LIN {X 0,Y 249.09,Z 614.452,A -85,B 0,C 180,E1 -19011.52,E2 -19011.52} C_VEL
LIN {X 0,Y 249.134,Z 614.451,A -85,B 0,C 180,E1 -19015.483,E2 -19015.483} C_VEL
LIN {X 0,Y 249.086,Z 614.457,A -85,B 0,C 180,E1 -19018.994,E2 -19018.994} C_VEL
LIN {X 0,Y 249.034,Z 614.454,A -85,B 0,C 180,E1 -19022.427,E2 -19022.427} C_VEL
LIN {X 0,Y 249.033,Z 614.454,A -85,B 0,C 180,E1 -19026.347,E2 -19026.347} C_VEL
LIN {X 0,Y 249.01,Z 614.463,A -85,B 0,C 180,E1 -19030.479,E2 -19030.479} C_VEL
LIN {X 0,Y 249.012,Z 614.464,A -85,B 0,C 180,E1 -19034.879,E2 -19034.879} C_VEL
LIN {X 0,Y 249.023,Z 614.461,A -85,B 0,C 180,E1 -19037.364,E2 -19037.364} C_VEL
LIN {X 0,Y 249.048,Z 614.442,A -85,B 0,C 180,E1 -19042.201,E2 -19042.201} C_VEL
LIN {X 0,Y 249.062,Z 614.452,A -85,B 0,C 180,E1 -19045.642,E2 -19045.642} C_VEL
LIN {X 0,Y 249.058,Z 614.459,A -85,B 0,C 180,E1 -19049.474,E2 -19049.474} C_VEL
LIN {X 0,Y 249.076,Z 614.457,A -85,B 0,C 180,E1 -19053.163,E2 -19053.163} C_VEL
LIN {X 0,Y 249.067,Z 614.455,A -85,B 0,C 180,E1 -19056.732,E2 -19056.732} C_VEL
LIN {X 0,Y 249.114,Z 614.444,A -85,B 0,C 180,E1 -19060.212,E2 -19060.212} C_VEL
LIN {X 0,Y 249.229,Z 614.424,A -85,B 0,C 180,E1 -19063.621,E2 -19063.621} C_VEL
LIN {X 0,Y 249.251,Z 614.432,A -85,B 0,C 180,E1 -19068.617,E2 -19068.617} C_VEL
LIN {X 0,Y 249.461,Z 614.411,A -85,B 0,C 180,E1 -19071.902,E2 -19071.902} C_VEL
LIN {X 0,Y 249.302,Z 614.427,A -85,B 0,C 180,E1 -19075.149,E2 -19075.149} C_VEL
LIN {X 0,Y 249.682,Z 614.378,A -85,B 0,C 180,E1 -19078.387,E2 -19078.387} C_VEL
LIN {X 0,Y 249.682,Z 614.371,A -85,B 0,C 180,E1 -19081.613,E2 -19081.613} C_VEL
LIN {X 0,Y 249.46,Z 614.411,A -85,B 0,C 180,E1 -19086.471,E2 -19086.471} C_VEL
LIN {X 0,Y 249.35,Z 614.423,A -85,B 0,C 180,E1 -19089.736,E2 -19089.736} C_VEL
LIN {X 0,Y 249.208,Z 614.436,A -85,B 0,C 180,E1 -19093.176,E2 -19093.176} C_VEL
LIN {X 0,Y 248.455,Z 614.531,A -85,B 0,C 180,E1 -19094.523,E2 -19094.523} C_VEL
LIN {X 0,Y 245.512,Z 614.901,A -85,B 0,C 180,E1 -19096.719,E2 -19096.719} C_VEL
LIN {X 0,Y 243.082,Z 615.206,A -85,B 0,C 180,E1 -19098.507,E2 -19098.507} C_VEL
LIN {X 0,Y 242.083,Z 615.329,A -85,B 0,C 180,E1 -19099.896,E2 -19099.896} C_VEL
LIN {X 0,Y 242.022,Z 615.339,A -85,B 0,C 180,E1 -19100.366,E2 -19100.366} C_VEL
LIN {X 0,Y 242.047,Z 615.332,A -85,B 0,C 180,E1 -19103.985,E2 -19103.985} C_VEL
LIN {X 0,Y 242.014,Z 615.337,A -85,B 0,C 180,E1 -19107.687,E2 -19107.687} C_VEL
LIN {X 0,Y 241.981,Z 615.34,A -85,B 0,C 180,E1 -19111.52,E2 -19111.52} C_VEL
LIN {X 0,Y 242.012,Z 615.337,A -85,B 0,C 180,E1 -19115.596,E2 -19115.596} C_VEL
LIN {X 0,Y 241.962,Z 615.344,A -85,B 0,C 180,E1 -19119.718,E2 -19119.718} C_VEL
LIN {X 0,Y 241.94,Z 615.348,A -85,B 0,C 180,E1 -19124.2,E2 -19124.2} C_VEL
LIN {X 0,Y 241.945,Z 615.346,A -85,B 0,C 180,E1 -19128.077,E2 -19128.077} C_VEL
LIN {X 0,Y 242.052,Z 615.51,A -85,B 0,C 180,E1 -19132.427,E2 -19132.427} C_VEL
LIN {X 0,Y 244.646,Z 627.471,A -85,B 0,C 180,E1 -19136.918,E2 -19136.918} C_VEL
LIN {X 0,Y 246.406,Z 636.286,A -85,B 0,C 180,E1 -19140.064,E2 -19140.064} C_VEL
LIN {X 0,Y 249.038,Z 644.626,A -85,B 0,C 180,E1 -19140.629,E2 -19140.629} C_VEL
LIN {X 0,Y 254.197,Z 690.653,A -85,B 0,C 180,E1 -19142.772,E2 -19142.772} C_VEL
LIN {X 0,Y 251.927,Z 745.701,A -85,B 0,C 180,E1 -19144.655,E2 -19144.655} C_VEL
LIN {X 0,Y 250.918,Z 759.315,A -85,B 0,C 180,E1 -19145.431,E2 -19145.431} C_VEL
LIN {X 0,Y 249.494,Z 771.741,A -85,B 0,C 180,E1 -19146.442,E2 -19146.442} C_VEL
LIN {X 0,Y 247.996,Z 783.383,A -85,B 0,C 180,E1 -19147.724,E2 -19147.724} C_VEL
LIN {X 0,Y 246.379,Z 794.75,A -85,B 0,C 180,E1 -19149.327,E2 -19149.327} C_VEL
LIN {X 0,Y 244.853,Z 805.07,A -85,B 0,C 180,E1 -19151.159,E2 -19151.159} C_VEL
LIN {X 0,Y 243.381,Z 814.349,A -85,B 0,C 180,E1 -19153.214,E2 -19153.214} C_VEL
LIN {X 0,Y 242.001,Z 823.396,A -85,B 0,C 180,E1 -19155.707,E2 -19155.707} C_VEL
LIN {X 0,Y 240.951,Z 830.593,A -85,B 0,C 180,E1 -19158.217,E2 -19158.217} C_VEL
LIN {X 0,Y 240.406,Z 836.316,A -85,B 0,C 180,E1 -19160.746,E2 -19160.746} C_VEL
LIN {X 0,Y 240.177,Z 840.763,A -85,B 0,C 180,E1 -19163.277,E2 -19163.277} C_VEL
LIN {X 0,Y 240.138,Z 843.082,A -85,B 0,C 180,E1 -19164.961,E2 -19164.961} C_VEL
LIN {X 0,Y 240.121,Z 844.923,A -85,B 0,C 180,E1 -19166.642,E2 -19166.642} C_VEL
LIN {X 0,Y 240.106,Z 846.259,A -85,B 0,C 180,E1 -19168.321,E2 -19168.321} C_VEL
LIN {X 0,Y 240.181,Z 847.174,A -85,B 0,C 180,E1 -19169.998,E2 -19169.998} C_VEL
LIN {X 0,Y 240.065,Z 847.656,A -85,B 0,C 180,E1 -19171.676,E2 -19171.676} C_VEL
LIN {X 0,Y 240,Z 847.701,A -85,B 0,C 180,E1 -19173.356,E2 -19173.356} C_VEL
LIN {X 0,Y 239.982,Z 846.513,A -85,B 0,C 180,E1 -19176.725,E2 -19176.725} C_VEL
LIN {X 0,Y 240.174,Z 845.328,A -85,B 0,C 180,E1 -19178.411,E2 -19178.411} C_VEL
LIN {X 0,Y 240.765,Z 842.736,A -85,B 0,C 180,E1 -19180.936,E2 -19180.936} C_VEL
LIN {X 0,Y 241.698,Z 839.154,A -85,B 0,C 180,E1 -19183.449,E2 -19183.449} C_VEL
LIN {X 0,Y 243.307,Z 834.5,A -85,B 0,C 180,E1 -19185.925,E2 -19185.925} C_VEL
LIN {X 0,Y 245.188,Z 828.664,A -85,B 0,C 180,E1 -19188.377,E2 -19188.377} C_VEL
LIN {X 0,Y 247.548,Z 821.5,A -85,B 0,C 180,E1 -19190.784,E2 -19190.784} C_VEL
LIN {X 0,Y 250.481,Z 812.616,A -85,B 0,C 180,E1 -19193.128,E2 -19193.128} C_VEL
LIN {X 0,Y 253.214,Z 803.619,A -85,B 0,C 180,E1 -19195.039,E2 -19195.039} C_VEL
LIN {X 0,Y 256.378,Z 792.642,A -85,B 0,C 180,E1 -19196.89,E2 -19196.89} C_VEL
LIN {X 0,Y 259.194,Z 781.744,A -85,B 0,C 180,E1 -19198.325,E2 -19198.325} C_VEL
LIN {X 0,Y 261.882,Z 769.864,A -85,B 0,C 180,E1 -19199.544,E2 -19199.544} C_VEL
LIN {X 0,Y 264.132,Z 757.818,A -85,B 0,C 180,E1 -19200.476,E2 -19200.476} C_VEL
LIN {X 0,Y 265.875,Z 744.095,A -85,B 0,C 180,E1 -19201.247,E2 -19201.247} C_VEL
LIN {X 0,Y 267.554,Z 722.588,A -85,B 0,C 180,E1 -19202.004,E2 -19202.004} C_VEL
LIN {X 0,Y 269.546,Z 692.623,A -85,B 0,C 180,E1 -19203.018,E2 -19203.018} C_VEL
LIN {X 0,Y 268.044,Z 675.513,A -85,B 0,C 180,E1 -19204.173,E2 -19204.173} C_VEL
LIN {X 0,Y 266.933,Z 667.783,A -85,B 0,C 180,E1 -19204.815,E2 -19204.815} C_VEL
LIN {X 0,Y 261.946,Z 656.396,A -85,B 0,C 180,E1 -19206.616,E2 -19206.616} C_VEL
LIN {X 0,Y 256.701,Z 646.257,A -85,B 0,C 180,E1 -19208.625,E2 -19208.625} C_VEL
LIN {X 0,Y 253.564,Z 640.832,A -85,B 0,C 180,E1 -19209.927,E2 -19209.927} C_VEL
LIN {X 0,Y 250.312,Z 635.27,A -85,B 0,C 180,E1 -19211.38,E2 -19211.38} C_VEL
LIN {X 0,Y 246.826,Z 629.984,A -85,B 0,C 180,E1 -19213.06,E2 -19213.06} C_VEL
LIN {X 0,Y 246.403,Z 629.005,A -85,B 0,C 180,E1 -19213.361,E2 -19213.361} C_VEL
LIN {X 0,Y 244.701,Z 623.368,A -85,B 0,C 180,E1 -19217.551,E2 -19217.551} C_VEL
LIN {X 0,Y 243.332,Z 619.435,A -85,B 0,C 180,E1 -19221.241,E2 -19221.241} C_VEL
LIN {X 0,Y 243.018,Z 618.149,A -85,B 0,C 180,E1 -19222.604,E2 -19222.604} C_VEL
LIN {X 0,Y 241.985,Z 615.336,A -85,B 0,C 180,E1 -19226.508,E2 -19226.508} C_VEL
LIN {X 0,Y 242.007,Z 615.332,A -85,B 0,C 180,E1 -19230.596,E2 -19230.596} C_VEL
LIN {X 0,Y 242.061,Z 615.323,A -85,B 0,C 180,E1 -19234.182,E2 -19234.182} C_VEL
LIN {X 0,Y 242.047,Z 615.336,A -85,B 0,C 180,E1 -19238.296,E2 -19238.296} C_VEL
LIN {X 0,Y 242.156,Z 615.318,A -85,B 0,C 180,E1 -19243.277,E2 -19243.277} C_VEL
LIN {X 0,Y 242.191,Z 615.438,A -85,B 0,C 180,E1 -19247.216,E2 -19247.216} C_VEL
LIN {X 0,Y 243.204,Z 617.796,A -85,B 0,C 180,E1 -19250.433,E2 -19250.433} C_VEL
LIN {X 0,Y 246.677,Z 622.197,A -85,B 0,C 180,E1 -19252.324,E2 -19252.324} C_VEL
LIN {X 0,Y 248.068,Z 623.799,A -85,B 0,C 180,E1 -19253.001,E2 -19253.001} C_VEL
LIN {X 0,Y 250.491,Z 627.155,A -85,B 0,C 180,E1 -19254.162,E2 -19254.162} C_VEL
LIN {X 0,Y 255.517,Z 633.633,A -85,B 0,C 180,E1 -19256.267,E2 -19256.267} C_VEL
LIN {X 0,Y 258.653,Z 638.212,A -85,B 0,C 180,E1 -19257.49,E2 -19257.49} C_VEL
LIN {X 0,Y 262.624,Z 644.888,A -85,B 0,C 180,E1 -19258.956,E2 -19258.956} C_VEL
LIN {X 0,Y 268.996,Z 656.761,A -85,B 0,C 180,E1 -19261.126,E2 -19261.126} C_VEL
LIN {X 0,Y 271.338,Z 662.521,A -85,B 0,C 180,E1 -19261.936,E2 -19261.936} C_VEL
LIN {X 0,Y 267.251,Z 720.175,A -85,B 0,C 180,E1 -19263.904,E2 -19263.904} C_VEL
LIN {X 0,Y 265.754,Z 733.662,A -85,B 0,C 180,E1 -19264.645,E2 -19264.645} C_VEL
LIN {X 0,Y 263.976,Z 746.003,A -85,B 0,C 180,E1 -19265.634,E2 -19265.634} C_VEL
LIN {X 0,Y 261.538,Z 758.402,A -85,B 0,C 180,E1 -19266.954,E2 -19266.954} C_VEL
LIN {X 0,Y 258.731,Z 770.225,A -85,B 0,C 180,E1 -19268.592,E2 -19268.592} C_VEL
LIN {X 0,Y 256.044,Z 780.215,A -85,B 0,C 180,E1 -19270.375,E2 -19270.375} C_VEL
LIN {X 0,Y 253.014,Z 789.597,A -85,B 0,C 180,E1 -19272.431,E2 -19272.431} C_VEL
LIN {X 0,Y 250.307,Z 797.53,A -85,B 0,C 180,E1 -19274.637,E2 -19274.637} C_VEL
LIN {X 0,Y 247.9,Z 803.973,A -85,B 0,C 180,E1 -19276.893,E2 -19276.893} C_VEL
LIN {X 0,Y 245.756,Z 809.422,A -85,B 0,C 180,E1 -19279.321,E2 -19279.321} C_VEL
LIN {X 0,Y 243.88,Z 814.004,A -85,B 0,C 180,E1 -19282.001,E2 -19282.001} C_VEL
LIN {X 0,Y 242.823,Z 816.492,A -85,B 0,C 180,E1 -19283.904,E2 -19283.904} C_VEL
LIN {X 0,Y 241.896,Z 818.362,A -85,B 0,C 180,E1 -19285.836,E2 -19285.836} C_VEL
LIN {X 0,Y 240.806,Z 820.184,A -85,B 0,C 180,E1 -19288.893,E2 -19288.893} C_VEL
LIN {X 0,Y 240.157,Z 820.642,A -85,B 0,C 180,E1 -19291.938,E2 -19291.938} C_VEL
LIN {X 0,Y 239.883,Z 819.775,A -85,B 0,C 180,E1 -19294.886,E2 -19294.886} C_VEL
LIN {X 0,Y 239.936,Z 817.519,A -85,B 0,C 180,E1 -19297.96,E2 -19297.96} C_VEL
LIN {X 0,Y 240.273,Z 814.563,A -85,B 0,C 180,E1 -19300.495,E2 -19300.495} C_VEL
LIN {X 0,Y 240.812,Z 810.309,A -85,B 0,C 180,E1 -19303.149,E2 -19303.149} C_VEL
LIN {X 0,Y 241.706,Z 804.016,A -85,B 0,C 180,E1 -19306.093,E2 -19306.093} C_VEL
LIN {X 0,Y 242.861,Z 796.483,A -85,B 0,C 180,E1 -19308.798,E2 -19308.798} C_VEL
LIN {X 0,Y 244.104,Z 788.762,A -85,B 0,C 180,E1 -19311.019,E2 -19311.019} C_VEL
LIN {X 0,Y 245.628,Z 779.186,A -85,B 0,C 180,E1 -19313.239,E2 -19313.239} C_VEL
LIN {X 0,Y 247.171,Z 769.108,A -85,B 0,C 180,E1 -19315.118,E2 -19315.118} C_VEL
LIN {X 0,Y 248.769,Z 757.73,A -85,B 0,C 180,E1 -19316.819,E2 -19316.819} C_VEL
LIN {X 0,Y 250.155,Z 745.895,A -85,B 0,C 180,E1 -19318.196,E2 -19318.196} C_VEL
LIN {X 0,Y 251.352,Z 732.633,A -85,B 0,C 180,E1 -19319.37,E2 -19319.37} C_VEL
LIN {X 0,Y 252.214,Z 719.571,A -85,B 0,C 180,E1 -19320.175,E2 -19320.175} C_VEL
LIN {X 0,Y 253.12,Z 698.707,A -85,B 0,C 180,E1 -19320.949,E2 -19320.949} C_VEL
LIN {X 0,Y 255.107,Z 648.228,A -85,B 0,C 180,E1 -19322.633,E2 -19322.633} C_VEL
LIN {X 0,Y 249.56,Z 633.732,A -85,B 0,C 180,E1 -19323.648,E2 -19323.648} C_VEL
LIN {X 0,Y 242.276,Z 616.171,A -85,B 0,C 180,E1 -19325.014,E2 -19325.014} C_VEL
LIN {X 0,Y 242.084,Z 615.328,A -85,B 0,C 180,E1 -19325.107,E2 -19325.107} C_VEL
LIN {X 0,Y 242.059,Z 615.334,A -85,B 0,C 180,E1 -19329.612,E2 -19329.612} C_VEL
LIN {X 0,Y 242.161,Z 615.318,A -85,B 0,C 180,E1 -19333.28,E2 -19333.28} C_VEL
LIN {X 0,Y 242.187,Z 615.319,A -85,B 0,C 180,E1 -19338.282,E2 -19338.282} C_VEL
LIN {X 0,Y 242.435,Z 615.285,A -85,B 0,C 180,E1 -19341.668,E2 -19341.668} C_VEL
LIN {X 0,Y 242.262,Z 615.307,A -85,B 0,C 180,E1 -19345.009,E2 -19345.009} C_VEL
LIN {X 0,Y 242.638,Z 615.263,A -85,B 0,C 180,E1 -19348.342,E2 -19348.342} C_VEL
LIN {X 0,Y 242.641,Z 615.259,A -85,B 0,C 180,E1 -19351.662,E2 -19351.662} C_VEL
LIN {X 0,Y 242.436,Z 615.287,A -85,B 0,C 180,E1 -19356.661,E2 -19356.661} C_VEL
LIN {X 0,Y 242.348,Z 615.295,A -85,B 0,C 180,E1 -19360.022,E2 -19360.022} C_VEL
LIN {X 0,Y 242.17,Z 615.318,A -85,B 0,C 180,E1 -19365.142,E2 -19365.142} C_VEL
LIN {X 0,Y 242.076,Z 615.327,A -85,B 0,C 180,E1 -19368.626,E2 -19368.626} C_VEL
LIN {X 0,Y 242.016,Z 615.333,A -85,B 0,C 180,E1 -19372.181,E2 -19372.181} C_VEL
LIN {X 0,Y 242.07,Z 615.329,A -85,B 0,C 180,E1 -19375.84,E2 -19375.84} C_VEL
LIN {X 0,Y 242.034,Z 615.331,A -85,B 0,C 180,E1 -19379.582,E2 -19379.582} C_VEL
LIN {X 0,Y 241.984,Z 615.327,A -85,B 0,C 180,E1 -19383.494,E2 -19383.494} C_VEL
LIN {X 0,Y 241.99,Z 615.337,A -85,B 0,C 180,E1 -19387.584,E2 -19387.584} C_VEL
LIN {X 0,Y 241.943,Z 615.345,A -85,B 0,C 180,E1 -19391.923,E2 -19391.923} C_VEL
LIN {X 0,Y 241.942,Z 615.341,A -85,B 0,C 180,E1 -19396.572,E2 -19396.572} C_VEL
LIN {X 0,Y 241.961,Z 615.33,A -85,B 0,C 180,E1 -19400.282,E2 -19400.282} C_VEL
LIN {X 0,Y 242.01,Z 615.324,A -85,B 0,C 180,E1 -19404.493,E2 -19404.493} C_VEL
LIN {X 0,Y 241.981,Z 615.337,A -85,B 0,C 180,E1 -19408.481,E2 -19408.481} C_VEL
LIN {X 0,Y 242.013,Z 615.337,A -85,B 0,C 180,E1 -19412.314,E2 -19412.314} C_VEL
LIN {X 0,Y 242.047,Z 615.332,A -85,B 0,C 180,E1 -19416.015,E2 -19416.015} C_VEL
LIN {X 0,Y 242.041,Z 615.329,A -85,B 0,C 180,E1 -19419.608,E2 -19419.608} C_VEL
LIN {X 0,Y 242.17,Z 615.301,A -85,B 0,C 180,E1 -19423.279,E2 -19423.279} C_VEL
LIN {X 0,Y 242.187,Z 615.313,A -85,B 0,C 180,E1 -19428.28,E2 -19428.28} C_VEL
LIN {X 0,Y 242.407,Z 615.288,A -85,B 0,C 180,E1 -19431.665,E2 -19431.665} C_VEL
LIN {X 0,Y 242.262,Z 615.304,A -85,B 0,C 180,E1 -19435.007,E2 -19435.007} C_VEL
LIN {X 0,Y 242.642,Z 615.254,A -85,B 0,C 180,E1 -19438.34,E2 -19438.34} C_VEL
LIN {X 0,Y 242.642,Z 615.247,A -85,B 0,C 180,E1 -19441.66,E2 -19441.66} C_VEL
LIN {X 0,Y 242.431,Z 615.285,A -85,B 0,C 180,E1 -19446.659,E2 -19446.659} C_VEL
LIN {X 0,Y 242.274,Z 615.306,A -85,B 0,C 180,E1 -19450.024,E2 -19450.024} C_VEL
LIN {X 0,Y 242.134,Z 615.315,A -85,B 0,C 180,E1 -19455.143,E2 -19455.143} C_VEL
LIN {X 0,Y 242.049,Z 615.336,A -85,B 0,C 180,E1 -19458.626,E2 -19458.626} C_VEL
LIN {X 0,Y 242.022,Z 615.339,A -85,B 0,C 180,E1 -19460.366,E2 -19460.366} C_VEL
LIN {X 0,Y 241.4,Z 615.424,A -85,B 0,C 180,E1 -19461.756,E2 -19461.756} C_VEL
LIN {X 0,Y 238.534,Z 615.777,A -85,B 0,C 180,E1 -19464.02,E2 -19464.02} C_VEL
LIN {X 0,Y 236.07,Z 616.077,A -85,B 0,C 180,E1 -19465.866,E2 -19465.866} C_VEL
LIN {X 0,Y 235.015,Z 616.21,A -85,B 0,C 180,E1 -19467.3,E2 -19467.3} C_VEL
LIN {X 0,Y 234.933,Z 616.217,A -85,B 0,C 180,E1 -19467.786,E2 -19467.786} C_VEL
LIN {X 0,Y 234.938,Z 616.223,A -85,B 0,C 180,E1 -19470.567,E2 -19470.567} C_VEL
LIN {X 0,Y 234.936,Z 616.22,A -85,B 0,C 180,E1 -19474.637,E2 -19474.637} C_VEL
LIN {X 0,Y 234.948,Z 616.221,A -85,B 0,C 180,E1 -19478.944,E2 -19478.944} C_VEL
LIN {X 0,Y 234.896,Z 616.226,A -85,B 0,C 180,E1 -19483.484,E2 -19483.484} C_VEL
LIN {X 0,Y 234.896,Z 616.226,A -85,B 0,C 180,E1 -19486.514,E2 -19486.514} C_VEL
LIN {X 0,Y 234.958,Z 616.218,A -85,B 0,C 180,E1 -19491.633,E2 -19491.633} C_VEL
LIN {X 0,Y 234.992,Z 616.275,A -85,B 0,C 180,E1 -19491.912,E2 -19491.912} C_VEL
LIN {X 0,Y 237.244,Z 626.919,A -85,B 0,C 180,E1 -19496.044,E2 -19496.044} C_VEL
LIN {X 0,Y 239.128,Z 636.083,A -85,B 0,C 180,E1 -19499.38,E2 -19499.38} C_VEL
LIN {X 0,Y 242.507,Z 646.258,A -85,B 0,C 180,E1 -19500.104,E2 -19500.104} C_VEL
LIN {X 0,Y 247.472,Z 690.694,A -85,B 0,C 180,E1 -19502.25,E2 -19502.25} C_VEL
LIN {X 0,Y 245.129,Z 745.513,A -85,B 0,C 180,E1 -19504.185,E2 -19504.185} C_VEL
LIN {X 0,Y 244.097,Z 759.046,A -85,B 0,C 180,E1 -19504.982,E2 -19504.982} C_VEL
LIN {X 0,Y 242.579,Z 771.91,A -85,B 0,C 180,E1 -19506.069,E2 -19506.069} C_VEL
LIN {X 0,Y 240.9,Z 784.211,A -85,B 0,C 180,E1 -19507.484,E2 -19507.484} C_VEL
LIN {X 0,Y 239.249,Z 795.356,A -85,B 0,C 180,E1 -19509.133,E2 -19509.133} C_VEL
LIN {X 0,Y 237.565,Z 806.32,A -85,B 0,C 180,E1 -19511.205,E2 -19511.205} C_VEL
LIN {X 0,Y 235.958,Z 816.257,A -85,B 0,C 180,E1 -19513.561,E2 -19513.561} C_VEL
LIN {X 0,Y 234.646,Z 824.795,A -85,B 0,C 180,E1 -19516.135,E2 -19516.135} C_VEL
LIN {X 0,Y 233.751,Z 831.643,A -85,B 0,C 180,E1 -19518.728,E2 -19518.728} C_VEL
LIN {X 0,Y 233.253,Z 837.07,A -85,B 0,C 180,E1 -19521.333,E2 -19521.333} C_VEL
LIN {X 0,Y 233.101,Z 841.65,A -85,B 0,C 180,E1 -19524.244,E2 -19524.244} C_VEL
LIN {X 0,Y 233.058,Z 844.256,A -85,B 0,C 180,E1 -19526.54,E2 -19526.54} C_VEL
LIN {X 0,Y 233.033,Z 845.674,A -85,B 0,C 180,E1 -19528.27,E2 -19528.27} C_VEL
LIN {X 0,Y 233.101,Z 846.634,A -85,B 0,C 180,E1 -19529.998,E2 -19529.998} C_VEL
LIN {X 0,Y 232.99,Z 847.159,A -85,B 0,C 180,E1 -19531.727,E2 -19531.727} C_VEL
LIN {X 0,Y 232.911,Z 847.276,A -85,B 0,C 180,E1 -19533.458,E2 -19533.458} C_VEL
LIN {X 0,Y 232.841,Z 846.949,A -85,B 0,C 180,E1 -19535.193,E2 -19535.193} C_VEL
LIN {X 0,Y 233.115,Z 845.072,A -85,B 0,C 180,E1 -19538.668,E2 -19538.668} C_VEL
LIN {X 0,Y 233.497,Z 843.536,A -85,B 0,C 180,E1 -19540.402,E2 -19540.402} C_VEL
LIN {X 0,Y 234.375,Z 840.387,A -85,B 0,C 180,E1 -19542.995,E2 -19542.995} C_VEL
LIN {X 0,Y 235.862,Z 836.23,A -85,B 0,C 180,E1 -19545.554,E2 -19545.554} C_VEL
LIN {X 0,Y 238.069,Z 829.963,A -85,B 0,C 180,E1 -19548.501,E2 -19548.501} C_VEL
LIN {X 0,Y 240.479,Z 823.171,A -85,B 0,C 180,E1 -19550.976,E2 -19550.976} C_VEL
LIN {X 0,Y 243.4,Z 814.814,A -85,B 0,C 180,E1 -19553.39,E2 -19553.39} C_VEL
LIN {X 0,Y 246.324,Z 806.382,A -85,B 0,C 180,E1 -19555.337,E2 -19555.337} C_VEL
LIN {X 0,Y 249.175,Z 797.33,A -85,B 0,C 180,E1 -19557.05,E2 -19557.05} C_VEL
LIN {X 0,Y 252.318,Z 786.286,A -85,B 0,C 180,E1 -19558.714,E2 -19558.714} C_VEL
LIN {X 0,Y 255.444,Z 773.963,A -85,B 0,C 180,E1 -19560.137,E2 -19560.137} C_VEL
LIN {X 0,Y 257.869,Z 762.16,A -85,B 0,C 180,E1 -19561.184,E2 -19561.184} C_VEL
LIN {X 0,Y 260.109,Z 747.995,A -85,B 0,C 180,E1 -19562.078,E2 -19562.078} C_VEL
LIN {X 0,Y 261.579,Z 733.711,A -85,B 0,C 180,E1 -19562.668,E2 -19562.668} C_VEL
LIN {X 0,Y 264.451,Z 693.887,A -85,B 0,C 180,E1 -19564.042,E2 -19564.042} C_VEL
LIN {X 0,Y 263.15,Z 677.789,A -85,B 0,C 180,E1 -19565.166,E2 -19565.166} C_VEL
LIN {X 0,Y 262.152,Z 670.998,A -85,B 0,C 180,E1 -19565.763,E2 -19565.763} C_VEL
LIN {X 0,Y 257.876,Z 660.878,A -85,B 0,C 180,E1 -19567.44,E2 -19567.44} C_VEL
LIN {X 0,Y 253.124,Z 651.404,A -85,B 0,C 180,E1 -19569.386,E2 -19569.386} C_VEL
LIN {X 0,Y 250.3,Z 646.33,A -85,B 0,C 180,E1 -19570.626,E2 -19570.626} C_VEL
LIN {X 0,Y 247.149,Z 640.848,A -85,B 0,C 180,E1 -19572.12,E2 -19572.12} C_VEL
LIN {X 0,Y 243.758,Z 635.331,A -85,B 0,C 180,E1 -19573.879,E2 -19573.879} C_VEL
LIN {X 0,Y 239.537,Z 629.3,A -85,B 0,C 180,E1 -19576.337,E2 -19576.337} C_VEL
LIN {X 0,Y 238.846,Z 627.89,A -85,B 0,C 180,E1 -19576.833,E2 -19576.833} C_VEL
LIN {X 0,Y 237.669,Z 624.13,A -85,B 0,C 180,E1 -19580.246,E2 -19580.246} C_VEL
LIN {X 0,Y 236.654,Z 621.209,A -85,B 0,C 180,E1 -19583.562,E2 -19583.562} C_VEL
LIN {X 0,Y 236.001,Z 619.137,A -85,B 0,C 180,E1 -19586.49,E2 -19586.49} C_VEL
LIN {X 0,Y 235.092,Z 616.975,A -85,B 0,C 180,E1 -19591.424,E2 -19591.424} C_VEL
LIN {X 0,Y 235.008,Z 616.205,A -85,B 0,C 180,E1 -19594.882,E2 -19594.882} C_VEL
LIN {X 0,Y 235.005,Z 616.222,A -85,B 0,C 180,E1 -19598.969,E2 -19598.969} C_VEL
LIN {X 0,Y 235.286,Z 617.222,A -85,B 0,C 180,E1 -19602.902,E2 -19602.902} C_VEL
LIN {X 0,Y 236.092,Z 618.98,A -85,B 0,C 180,E1 -19606.716,E2 -19606.716} C_VEL
LIN {X 0,Y 238.744,Z 622.515,A -85,B 0,C 180,E1 -19608.646,E2 -19608.646} C_VEL
LIN {X 0,Y 241.151,Z 624.593,A -85,B 0,C 180,E1 -19610.07,E2 -19610.07} C_VEL
LIN {X 0,Y 244.476,Z 628.746,A -85,B 0,C 180,E1 -19611.944,E2 -19611.944} C_VEL
LIN {X 0,Y 246.301,Z 631.399,A -85,B 0,C 180,E1 -19612.89,E2 -19612.89} C_VEL
LIN {X 0,Y 249.219,Z 635.19,A -85,B 0,C 180,E1 -19614.278,E2 -19614.278} C_VEL
LIN {X 0,Y 252.66,Z 639.789,A -85,B 0,C 180,E1 -19615.755,E2 -19615.755} C_VEL
LIN {X 0,Y 256.339,Z 645.372,A -85,B 0,C 180,E1 -19617.262,E2 -19617.262} C_VEL
LIN {X 0,Y 263.166,Z 658.178,A -85,B 0,C 180,E1 -19619.842,E2 -19619.842} C_VEL
LIN {X 0,Y 266.218,Z 664.61,A -85,B 0,C 180,E1 -19620.898,E2 -19620.898} C_VEL
LIN {X 0,Y 261.994,Z 721.142,A -85,B 0,C 180,E1 -19622.892,E2 -19622.892} C_VEL
LIN {X 0,Y 260.338,Z 734.926,A -85,B 0,C 180,E1 -19623.678,E2 -19623.678} C_VEL
LIN {X 0,Y 258.256,Z 748.052,A -85,B 0,C 180,E1 -19624.78,E2 -19624.78} C_VEL
LIN {X 0,Y 255.739,Z 760.064,A -85,B 0,C 180,E1 -19626.113,E2 -19626.113} C_VEL
LIN {X 0,Y 253.124,Z 770.531,A -85,B 0,C 180,E1 -19627.601,E2 -19627.601} C_VEL
LIN {X 0,Y 250.474,Z 779.913,A -85,B 0,C 180,E1 -19629.284,E2 -19629.284} C_VEL
LIN {X 0,Y 247.79,Z 787.852,A -85,B 0,C 180,E1 -19630.996,E2 -19630.996} C_VEL
LIN {X 0,Y 244.723,Z 796.298,A -85,B 0,C 180,E1 -19633.282,E2 -19633.282} C_VEL
LIN {X 0,Y 242.025,Z 803.245,A -85,B 0,C 180,E1 -19635.642,E2 -19635.642} C_VEL
LIN {X 0,Y 239.771,Z 808.574,A -85,B 0,C 180,E1 -19637.925,E2 -19637.925} C_VEL
LIN {X 0,Y 237.577,Z 813.692,A -85,B 0,C 180,E1 -19640.792,E2 -19640.792} C_VEL
LIN {X 0,Y 235.837,Z 817.379,A -85,B 0,C 180,E1 -19643.721,E2 -19643.721} C_VEL
LIN {X 0,Y 234.434,Z 819.811,A -85,B 0,C 180,E1 -19646.723,E2 -19646.723} C_VEL
LIN {X 0,Y 233.621,Z 820.875,A -85,B 0,C 180,E1 -19649.265,E2 -19649.265} C_VEL
LIN {X 0,Y 233.004,Z 820.961,A -85,B 0,C 180,E1 -19652.38,E2 -19652.38} C_VEL
LIN {X 0,Y 232.763,Z 819.795,A -85,B 0,C 180,E1 -19655.393,E2 -19655.393} C_VEL
LIN {X 0,Y 232.882,Z 817.459,A -85,B 0,C 180,E1 -19658.316,E2 -19658.316} C_VEL
LIN {X 0,Y 233.364,Z 813.444,A -85,B 0,C 180,E1 -19661.495,E2 -19661.495} C_VEL
LIN {X 0,Y 233.925,Z 809.401,A -85,B 0,C 180,E1 -19663.862,E2 -19663.862} C_VEL
LIN {X 0,Y 234.848,Z 802.822,A -85,B 0,C 180,E1 -19666.837,E2 -19666.837} C_VEL
LIN {X 0,Y 235.979,Z 795.789,A -85,B 0,C 180,E1 -19669.331,E2 -19669.331} C_VEL
LIN {X 0,Y 237.396,Z 787.283,A -85,B 0,C 180,E1 -19671.737,E2 -19671.737} C_VEL
LIN {X 0,Y 239.019,Z 777.426,A -85,B 0,C 180,E1 -19673.982,E2 -19673.982} C_VEL
LIN {X 0,Y 240.657,Z 766.648,A -85,B 0,C 180,E1 -19675.943,E2 -19675.943} C_VEL
LIN {X 0,Y 242.216,Z 755.048,A -85,B 0,C 180,E1 -19677.611,E2 -19677.611} C_VEL
LIN {X 0,Y 243.677,Z 743.022,A -85,B 0,C 180,E1 -19678.958,E2 -19678.958} C_VEL
LIN {X 0,Y 244.871,Z 729.452,A -85,B 0,C 180,E1 -19680.079,E2 -19680.079} C_VEL
LIN {X 0,Y 245.655,Z 716,A -85,B 0,C 180,E1 -19680.846,E2 -19680.846} C_VEL
LIN {X 0,Y 248.481,Z 649.907,A -85,B 0,C 180,E1 -19683.13,E2 -19683.13} C_VEL
LIN {X 0,Y 242.604,Z 634.793,A -85,B 0,C 180,E1 -19684.246,E2 -19684.246} C_VEL
LIN {X 0,Y 235.172,Z 617.035,A -85,B 0,C 180,E1 -19685.681,E2 -19685.681} C_VEL
LIN {X 0,Y 235.026,Z 616.209,A -85,B 0,C 180,E1 -19685.783,E2 -19685.783} C_VEL
LIN {X 0,Y 235.026,Z 616.209,A -85,B 0,C 180,E1 -19688.973,E2 -19688.973} C_VEL
LIN {X 0,Y 235.095,Z 616.198,A -85,B 0,C 180,E1 -19693.061,E2 -19693.061} C_VEL
LIN {X 0,Y 235.147,Z 616.194,A -85,B 0,C 180,E1 -19697.926,E2 -19697.926} C_VEL
LIN {X 0,Y 235.39,Z 616.163,A -85,B 0,C 180,E1 -19701.416,E2 -19701.416} C_VEL
LIN {X 0,Y 235.406,Z 616.161,A -85,B 0,C 180,E1 -19703.143,E2 -19703.143} C_VEL
LIN {X 0,Y 235.597,Z 616.14,A -85,B 0,C 180,E1 -19708.292,E2 -19708.292} C_VEL
LIN {X 0,Y 235.6,Z 616.136,A -85,B 0,C 180,E1 -19711.711,E2 -19711.711} C_VEL
LIN {X 0,Y 235.408,Z 616.162,A -85,B 0,C 180,E1 -19716.86,E2 -19716.86} C_VEL
LIN {X 0,Y 235.256,Z 616.18,A -85,B 0,C 180,E1 -19720.328,E2 -19720.328} C_VEL
LIN {X 0,Y 235.117,Z 616.195,A -85,B 0,C 180,E1 -19725.608,E2 -19725.608} C_VEL
LIN {X 0,Y 235.012,Z 616.201,A -85,B 0,C 180,E1 -19729.207,E2 -19729.207} C_VEL
LIN {X 0,Y 234.964,Z 616.214,A -85,B 0,C 180,E1 -19732.884,E2 -19732.884} C_VEL
LIN {X 0,Y 234.973,Z 616.215,A -85,B 0,C 180,E1 -19736.659,E2 -19736.659} C_VEL
LIN {X 0,Y 234.935,Z 616.215,A -85,B 0,C 180,E1 -19740.569,E2 -19740.569} C_VEL
LIN {X 0,Y 234.931,Z 616.203,A -85,B 0,C 180,E1 -19744.64,E2 -19744.64} C_VEL
LIN {X 0,Y 234.946,Z 616.214,A -85,B 0,C 180,E1 -19748.946,E2 -19748.946} C_VEL
LIN {X 0,Y 234.894,Z 616.225,A -85,B 0,C 180,E1 -19753.487,E2 -19753.487} C_VEL
LIN {X 0,Y 234.895,Z 616.219,A -85,B 0,C 180,E1 -19756.516,E2 -19756.516} C_VEL
LIN {X 0,Y 234.923,Z 616.207,A -85,B 0,C 180,E1 -19761.08,E2 -19761.08} C_VEL
LIN {X 0,Y 234.947,Z 616.205,A -85,B 0,C 180,E1 -19765.365,E2 -19765.365} C_VEL
LIN {X 0,Y 234.938,Z 616.217,A -85,B 0,C 180,E1 -19769.433,E2 -19769.433} C_VEL
LIN {X 0,Y 235,Z 616.213,A -85,B 0,C 180,E1 -19773.795,E2 -19773.795} C_VEL
LIN {X 0,Y 235.004,Z 616.203,A -85,B 0,C 180,E1 -19778.969,E2 -19778.969} C_VEL
LIN {X 0,Y 235.102,Z 616.179,A -85,B 0,C 180,E1 -19783.061,E2 -19783.061} C_VEL
LIN {X 0,Y 235.12,Z 616.19,A -85,B 0,C 180,E1 -19787.923,E2 -19787.923} C_VEL
LIN {X 0,Y 235.338,Z 616.167,A -85,B 0,C 180,E1 -19791.413,E2 -19791.413} C_VEL
LIN {X 0,Y 235.38,Z 616.162,A -85,B 0,C 180,E1 -19793.141,E2 -19793.141} C_VEL
LIN {X 0,Y 235.602,Z 616.131,A -85,B 0,C 180,E1 -19798.291,E2 -19798.291} C_VEL
LIN {X 0,Y 235.602,Z 616.123,A -85,B 0,C 180,E1 -19801.71,E2 -19801.71} C_VEL
LIN {X 0,Y 235.381,Z 616.163,A -85,B 0,C 180,E1 -19806.86,E2 -19806.86} C_VEL
LIN {X 0,Y 235.221,Z 616.187,A -85,B 0,C 180,E1 -19810.327,E2 -19810.327} C_VEL
LIN {X 0,Y 235.081,Z 616.193,A -85,B 0,C 180,E1 -19815.609,E2 -19815.609} C_VEL
LIN {X 0,Y 234.966,Z 616.213,A -85,B 0,C 180,E1 -19820.375,E2 -19820.375} C_VEL
LIN {X 0,Y 234.985,Z 616.211,A -85,B 0,C 180,E1 -19824.754,E2 -19824.754} C_VEL
LIN {X 0,Y 234.933,Z 616.217,A -85,B 0,C 180,E1 -19827.786,E2 -19827.786} C_VEL
LIN {X 0,Y 234.261,Z 616.306,A -85,B 0,C 180,E1 -19829.216,E2 -19829.216} C_VEL
LIN {X 0,Y 231.367,Z 616.662,A -85,B 0,C 180,E1 -19831.547,E2 -19831.547} C_VEL
LIN {X 0,Y 228.93,Z 616.966,A -85,B 0,C 180,E1 -19833.448,E2 -19833.448} C_VEL
LIN {X 0,Y 227.922,Z 617.096,A -85,B 0,C 180,E1 -19834.925,E2 -19834.925} C_VEL
LIN {X 0,Y 227.86,Z 617.096,A -85,B 0,C 180,E1 -19835.426,E2 -19835.426} C_VEL
LIN {X 0,Y 227.859,Z 617.102,A -85,B 0,C 180,E1 -19839.545,E2 -19839.545} C_VEL
LIN {X 0,Y 227.819,Z 617.11,A -85,B 0,C 180,E1 -19842.741,E2 -19842.741} C_VEL
LIN {X 0,Y 227.818,Z 617.108,A -85,B 0,C 180,E1 -19847.257,E2 -19847.257} C_VEL
LIN {X 0,Y 227.952,Z 617.281,A -85,B 0,C 180,E1 -19851.473,E2 -19851.473} C_VEL
LIN {X 0,Y 230.127,Z 627.438,A -85,B 0,C 180,E1 -19855.546,E2 -19855.546} C_VEL
LIN {X 0,Y 231.754,Z 635.399,A -85,B 0,C 180,E1 -19858.599,E2 -19858.599} C_VEL
LIN {X 0,Y 236.087,Z 648.824,A -85,B 0,C 180,E1 -19859.606,E2 -19859.606} C_VEL
LIN {X 0,Y 240.753,Z 691.576,A -85,B 0,C 180,E1 -19861.73,E2 -19861.73} C_VEL
LIN {X 0,Y 238.349,Z 745.324,A -85,B 0,C 180,E1 -19863.689,E2 -19863.689} C_VEL
LIN {X 0,Y 237.22,Z 759.486,A -85,B 0,C 180,E1 -19864.557,E2 -19864.557} C_VEL
LIN {X 0,Y 235.823,Z 771.113,A -85,B 0,C 180,E1 -19865.573,E2 -19865.573} C_VEL
LIN {X 0,Y 234.085,Z 783.484,A -85,B 0,C 180,E1 -19867.025,E2 -19867.025} C_VEL
LIN {X 0,Y 232.392,Z 794.694,A -85,B 0,C 180,E1 -19868.719,E2 -19868.719} C_VEL
LIN {X 0,Y 230.998,Z 803.841,A -85,B 0,C 180,E1 -19870.446,E2 -19870.446} C_VEL
LIN {X 0,Y 229.409,Z 813.199,A -85,B 0,C 180,E1 -19872.619,E2 -19872.619} C_VEL
LIN {X 0,Y 227.964,Z 822.311,A -85,B 0,C 180,E1 -19875.263,E2 -19875.263} C_VEL
LIN {X 0,Y 226.85,Z 829.568,A -85,B 0,C 180,E1 -19877.927,E2 -19877.927} C_VEL
LIN {X 0,Y 226.213,Z 836.151,A -85,B 0,C 180,E1 -19881.062,E2 -19881.062} C_VEL
LIN {X 0,Y 226.051,Z 839.161,A -85,B 0,C 180,E1 -19882.854,E2 -19882.854} C_VEL
LIN {X 0,Y 226.012,Z 841.595,A -85,B 0,C 180,E1 -19884.645,E2 -19884.645} C_VEL
LIN {X 0,Y 225.996,Z 843.552,A -85,B 0,C 180,E1 -19886.432,E2 -19886.432} C_VEL
LIN {X 0,Y 225.963,Z 845.055,A -85,B 0,C 180,E1 -19888.216,E2 -19888.216} C_VEL
LIN {X 0,Y 226.022,Z 846.078,A -85,B 0,C 180,E1 -19889.998,E2 -19889.998} C_VEL
LIN {X 0,Y 225.916,Z 846.655,A -85,B 0,C 180,E1 -19891.781,E2 -19891.781} C_VEL
LIN {X 0,Y 225.778,Z 846.637,A -85,B 0,C 180,E1 -19895.062,E2 -19895.062} C_VEL
LIN {X 0,Y 225.828,Z 845.903,A -85,B 0,C 180,E1 -19897.149,E2 -19897.149} C_VEL
LIN {X 0,Y 226.492,Z 843.34,A -85,B 0,C 180,E1 -19900.728,E2 -19900.728} C_VEL
LIN {X 0,Y 227.427,Z 840.321,A -85,B 0,C 180,E1 -19903.399,E2 -19903.399} C_VEL
LIN {X 0,Y 229.016,Z 836.289,A -85,B 0,C 180,E1 -19906.031,E2 -19906.031} C_VEL
LIN {X 0,Y 230.977,Z 831.146,A -85,B 0,C 180,E1 -19908.63,E2 -19908.63} C_VEL
LIN {X 0,Y 233.418,Z 824.763,A -85,B 0,C 180,E1 -19911.178,E2 -19911.178} C_VEL
LIN {X 0,Y 236.4,Z 816.963,A -85,B 0,C 180,E1 -19913.66,E2 -19913.66} C_VEL
LIN {X 0,Y 239.986,Z 807.272,A -85,B 0,C 180,E1 -19916.055,E2 -19916.055} C_VEL
LIN {X 0,Y 242.936,Z 798.468,A -85,B 0,C 180,E1 -19917.804,E2 -19917.804} C_VEL
LIN {X 0,Y 246.176,Z 787.839,A -85,B 0,C 180,E1 -19919.5,E2 -19919.5} C_VEL
LIN {X 0,Y 249.415,Z 776.097,A -85,B 0,C 180,E1 -19920.945,E2 -19920.945} C_VEL
LIN {X 0,Y 252.362,Z 762.964,A -85,B 0,C 180,E1 -19922.18,E2 -19922.18} C_VEL
LIN {X 0,Y 254.724,Z 749.569,A -85,B 0,C 180,E1 -19923.076,E2 -19923.076} C_VEL
LIN {X 0,Y 256.35,Z 735.923,A -85,B 0,C 180,E1 -19923.689,E2 -19923.689} C_VEL
LIN {X 0,Y 259.42,Z 694.621,A -85,B 0,C 180,E1 -19925.154,E2 -19925.154} C_VEL
LIN {X 0,Y 258.4,Z 680.292,A -85,B 0,C 180,E1 -19926.186,E2 -19926.186} C_VEL
LIN {X 0,Y 257.588,Z 674.296,A -85,B 0,C 180,E1 -19926.738,E2 -19926.738} C_VEL
LIN {X 0,Y 253.13,Z 663.876,A -85,B 0,C 180,E1 -19928.589,E2 -19928.589} C_VEL
LIN {X 0,Y 249.443,Z 656.226,A -85,B 0,C 180,E1 -19930.251,E2 -19930.251} C_VEL
LIN {X 0,Y 246.885,Z 651.555,A -85,B 0,C 180,E1 -19931.434,E2 -19931.434} C_VEL
LIN {X 0,Y 244.194,Z 646.596,A -85,B 0,C 180,E1 -19932.822,E2 -19932.822} C_VEL
LIN {X 0,Y 240.449,Z 640.463,A -85,B 0,C 180,E1 -19934.896,E2 -19934.896} C_VEL
LIN {X 0,Y 236.886,Z 634.936,A -85,B 0,C 180,E1 -19937.159,E2 -19937.159} C_VEL
LIN {X 0,Y 235.662,Z 633.195,A -85,B 0,C 180,E1 -19938.023,E2 -19938.023} C_VEL
LIN {X 0,Y 231.042,Z 626.18,A -85,B 0,C 180,E1 -19942.133,E2 -19942.133} C_VEL
LIN {X 0,Y 230.001,Z 622.914,A -85,B 0,C 180,E1 -19946.632,E2 -19946.632} C_VEL
LIN {X 0,Y 229.214,Z 621.141,A -85,B 0,C 180,E1 -19950.621,E2 -19950.621} C_VEL
LIN {X 0,Y 229.082,Z 620.107,A -85,B 0,C 180,E1 -19954.563,E2 -19954.563} C_VEL
LIN {X 0,Y 229.039,Z 620.031,A -85,B 0,C 180,E1 -19958.394,E2 -19958.394} C_VEL
LIN {X 0,Y 229.225,Z 620.771,A -85,B 0,C 180,E1 -19961.382,E2 -19961.382} C_VEL
LIN {X 0,Y 233.26,Z 625.015,A -85,B 0,C 180,E1 -19965.562,E2 -19965.562} C_VEL
LIN {X 0,Y 234.469,Z 626.09,A -85,B 0,C 180,E1 -19966.512,E2 -19966.512} C_VEL
LIN {X 0,Y 237.106,Z 629.435,A -85,B 0,C 180,E1 -19968.458,E2 -19968.458} C_VEL
LIN {X 0,Y 239.004,Z 631.126,A -85,B 0,C 180,E1 -19969.624,E2 -19969.624} C_VEL
LIN {X 0,Y 242.849,Z 636.213,A -85,B 0,C 180,E1 -19971.87,E2 -19971.87} C_VEL
LIN {X 0,Y 246.8,Z 641.745,A -85,B 0,C 180,E1 -19973.86,E2 -19973.86} C_VEL
LIN {X 0,Y 249.931,Z 646.106,A -85,B 0,C 180,E1 -19975.282,E2 -19975.282} C_VEL
LIN {X 0,Y 253.015,Z 650.964,A -85,B 0,C 180,E1 -19976.6,E2 -19976.6} C_VEL
LIN {X 0,Y 258.488,Z 661.506,A -85,B 0,C 180,E1 -19978.809,E2 -19978.809} C_VEL
LIN {X 0,Y 261.192,Z 667.187,A -85,B 0,C 180,E1 -19979.841,E2 -19979.841} C_VEL
LIN {X 0,Y 256.995,Z 720.949,A -85,B 0,C 180,E1 -19981.763,E2 -19981.763} C_VEL
LIN {X 0,Y 255.47,Z 733.539,A -85,B 0,C 180,E1 -19982.463,E2 -19982.463} C_VEL
LIN {X 0,Y 253.298,Z 747.149,A -85,B 0,C 180,E1 -19983.578,E2 -19983.578} C_VEL
LIN {X 0,Y 250.81,Z 758.575,A -85,B 0,C 180,E1 -19984.822,E2 -19984.822} C_VEL
LIN {X 0,Y 247.592,Z 770.838,A -85,B 0,C 180,E1 -19986.561,E2 -19986.561} C_VEL
LIN {X 0,Y 244.791,Z 780.194,A -85,B 0,C 180,E1 -19988.253,E2 -19988.253} C_VEL
LIN {X 0,Y 241.224,Z 790.148,A -85,B 0,C 180,E1 -19990.491,E2 -19990.491} C_VEL
LIN {X 0,Y 237.95,Z 798.593,A -85,B 0,C 180,E1 -19992.932,E2 -19992.932} C_VEL
LIN {X 0,Y 234.85,Z 805.769,A -85,B 0,C 180,E1 -19995.624,E2 -19995.624} C_VEL
LIN {X 0,Y 232.146,Z 811.68,A -85,B 0,C 180,E1 -19998.534,E2 -19998.534} C_VEL
LIN {X 0,Y 229.982,Z 816.114,A -85,B 0,C 180,E1 -20001.512,E2 -20001.512} C_VEL
LIN {X 0,Y 228.841,Z 818.279,A -85,B 0,C 180,E1 -20003.531,E2 -20003.531} C_VEL
LIN {X 0,Y 227.477,Z 820.387,A -85,B 0,C 180,E1 -20006.372,E2 -20006.372} C_VEL
LIN {X 0,Y 226.415,Z 821.512,A -85,B 0,C 180,E1 -20009.778,E2 -20009.778} C_VEL
LIN {X 0,Y 225.862,Z 821.221,A -85,B 0,C 180,E1 -20012.849,E2 -20012.849} C_VEL
LIN {X 0,Y 225.664,Z 819.466,A -85,B 0,C 180,E1 -20016.28,E2 -20016.28} C_VEL
LIN {X 0,Y 225.962,Z 816.083,A -85,B 0,C 180,E1 -20019.772,E2 -20019.772} C_VEL
LIN {X 0,Y 226.591,Z 811.302,A -85,B 0,C 180,E1 -20023.028,E2 -20023.028} C_VEL
LIN {X 0,Y 227.401,Z 805.807,A -85,B 0,C 180,E1 -20025.824,E2 -20025.824} C_VEL
LIN {X 0,Y 228.32,Z 799.805,A -85,B 0,C 180,E1 -20028.247,E2 -20028.247} C_VEL
LIN {X 0,Y 229.723,Z 791.517,A -85,B 0,C 180,E1 -20030.923,E2 -20030.923} C_VEL
LIN {X 0,Y 231.268,Z 782.434,A -85,B 0,C 180,E1 -20033.273,E2 -20033.273} C_VEL
LIN {X 0,Y 232.948,Z 772.199,A -85,B 0,C 180,E1 -20035.405,E2 -20035.405} C_VEL
LIN {X 0,Y 234.716,Z 760.718,A -85,B 0,C 180,E1 -20037.291,E2 -20037.291} C_VEL
LIN {X 0,Y 236.236,Z 748.493,A -85,B 0,C 180,E1 -20038.877,E2 -20038.877} C_VEL
LIN {X 0,Y 237.632,Z 735.19,A -85,B 0,C 180,E1 -20040.158,E2 -20040.158} C_VEL
LIN {X 0,Y 238.586,Z 722.021,A -85,B 0,C 180,E1 -20041.074,E2 -20041.074} C_VEL
LIN {X 0,Y 239.424,Z 705.129,A -85,B 0,C 180,E1 -20041.781,E2 -20041.781} C_VEL
LIN {X 0,Y 241.786,Z 651.361,A -85,B 0,C 180,E1 -20043.672,E2 -20043.672} C_VEL
LIN {X 0,Y 233.054,Z 629.331,A -85,B 0,C 180,E1 -20045.389,E2 -20045.389} C_VEL
LIN {X 0,Y 228.068,Z 617.796,A -85,B 0,C 180,E1 -20046.387,E2 -20046.387} C_VEL
LIN {X 0,Y 227.965,Z 617.09,A -85,B 0,C 180,E1 -20046.468,E2 -20046.468} C_VEL
LIN {X 0,Y 227.953,Z 617.09,A -85,B 0,C 180,E1 -20050.178,E2 -20050.178} C_VEL
LIN {X 0,Y 228.057,Z 617.076,A -85,B 0,C 180,E1 -20053.9,E2 -20053.9} C_VEL
LIN {X 0,Y 228.171,Z 617.061,A -85,B 0,C 180,E1 -20059.352,E2 -20059.352} C_VEL
LIN {X 0,Y 228.359,Z 617.04,A -85,B 0,C 180,E1 -20062.931,E2 -20062.931} C_VEL
LIN {X 0,Y 228.556,Z 617.016,A -85,B 0,C 180,E1 -20068.24,E2 -20068.24} C_VEL
LIN {X 0,Y 228.559,Z 617.013,A -85,B 0,C 180,E1 -20071.764,E2 -20071.764} C_VEL
LIN {X 0,Y 228.36,Z 617.038,A -85,B 0,C 180,E1 -20077.073,E2 -20077.073} C_VEL
LIN {X 0,Y 228.174,Z 617.063,A -85,B 0,C 180,E1 -20080.652,E2 -20080.652} C_VEL
LIN {X 0,Y 228.06,Z 617.074,A -85,B 0,C 180,E1 -20086.104,E2 -20086.104} C_VEL
LIN {X 0,Y 227.946,Z 617.078,A -85,B 0,C 180,E1 -20089.827,E2 -20089.827} C_VEL
LIN {X 0,Y 227.918,Z 617.092,A -85,B 0,C 180,E1 -20093.634,E2 -20093.634} C_VEL
LIN {X 0,Y 227.89,Z 617.096,A -85,B 0,C 180,E1 -20097.556,E2 -20097.556} C_VEL
LIN {X 0,Y 227.874,Z 617.089,A -85,B 0,C 180,E1 -20101.624,E2 -20101.624} C_VEL
LIN {X 0,Y 227.884,Z 617.087,A -85,B 0,C 180,E1 -20105.873,E2 -20105.873} C_VEL
LIN {X 0,Y 227.831,Z 617.101,A -85,B 0,C 180,E1 -20110.378,E2 -20110.378} C_VEL
LIN {X 0,Y 227.84,Z 617.103,A -85,B 0,C 180,E1 -20115.193,E2 -20115.193} C_VEL
LIN {X 0,Y 227.831,Z 617.091,A -85,B 0,C 180,E1 -20119.625,E2 -20119.625} C_VEL
LIN {X 0,Y 227.888,Z 617.081,A -85,B 0,C 180,E1 -20124.13,E2 -20124.13} C_VEL
LIN {X 0,Y 227.877,Z 617.093,A -85,B 0,C 180,E1 -20128.379,E2 -20128.379} C_VEL
LIN {X 0,Y 227.892,Z 617.096,A -85,B 0,C 180,E1 -20132.446,E2 -20132.446} C_VEL
LIN {X 0,Y 227.913,Z 617.091,A -85,B 0,C 180,E1 -20136.367,E2 -20136.367} C_VEL
LIN {X 0,Y 227.943,Z 617.079,A -85,B 0,C 180,E1 -20140.175,E2 -20140.175} C_VEL
LIN {X 0,Y 228.06,Z 617.056,A -85,B 0,C 180,E1 -20143.898,E2 -20143.898} C_VEL
LIN {X 0,Y 228.078,Z 617.064,A -85,B 0,C 180,E1 -20147.544,E2 -20147.544} C_VEL
LIN {X 0,Y 228.274,Z 617.046,A -85,B 0,C 180,E1 -20151.145,E2 -20151.145} C_VEL
LIN {X 0,Y 228.331,Z 617.04,A -85,B 0,C 180,E1 -20152.928,E2 -20152.928} C_VEL
LIN {X 0,Y 228.561,Z 617.008,A -85,B 0,C 180,E1 -20158.238,E2 -20158.238} C_VEL
LIN {X 0,Y 228.561,Z 616.999,A -85,B 0,C 180,E1 -20161.762,E2 -20161.762} C_VEL
LIN {X 0,Y 228.331,Z 617.04,A -85,B 0,C 180,E1 -20167.072,E2 -20167.072} C_VEL
LIN {X 0,Y 228.152,Z 617.065,A -85,B 0,C 180,E1 -20170.651,E2 -20170.651} C_VEL
LIN {X 0,Y 228.048,Z 617.073,A -85,B 0,C 180,E1 -20174.273,E2 -20174.273} C_VEL
LIN {X 0,Y 227.958,Z 617.086,A -85,B 0,C 180,E1 -20177.957,E2 -20177.957} C_VEL
LIN {X 0,Y 227.922,Z 617.096,A -85,B 0,C 180,E1 -20182.32,E2 -20182.32} C_VEL
LIN {X 0,Y 227.95,Z 617.089,A -85,B 0,C 180,E1 -20186.602,E2 -20186.602} C_VEL
LIN {X 0,Y 227.915,Z 617.096,A -85,B 0,C 180,E1 -20190.295,E2 -20190.295} C_VEL
LIN {X 0,Y 227.884,Z 617.095,A -85,B 0,C 180,E1 -20193.72,E2 -20193.72} C_VEL
LIN {X 0,Y 227.86,Z 617.096,A -85,B 0,C 180,E1 -20195.426,E2 -20195.426} C_VEL
LIN {X 0,Y 227.242,Z 617.182,A -85,B 0,C 180,E1 -20196.901,E2 -20196.901} C_VEL
LIN {X 0,Y 224.39,Z 617.545,A -85,B 0,C 180,E1 -20199.307,E2 -20199.307} C_VEL
LIN {X 0,Y 221.925,Z 617.851,A -85,B 0,C 180,E1 -20201.271,E2 -20201.271} C_VEL
LIN {X 0,Y 220.853,Z 617.979,A -85,B 0,C 180,E1 -20202.797,E2 -20202.797} C_VEL
LIN {X 0,Y 220.761,Z 617.988,A -85,B 0,C 180,E1 -20203.315,E2 -20203.315} C_VEL
LIN {X 0,Y 220.774,Z 617.986,A -85,B 0,C 180,E1 -20207.069,E2 -20207.069} C_VEL
LIN {X 0,Y 220.884,Z 618.083,A -85,B 0,C 180,E1 -20210.936,E2 -20210.936} C_VEL
LIN {X 0,Y 223.013,Z 627.926,A -85,B 0,C 180,E1 -20215.021,E2 -20215.021} C_VEL
LIN {X 0,Y 224.515,Z 635.21,A -85,B 0,C 180,E1 -20217.881,E2 -20217.881} C_VEL
LIN {X 0,Y 229.584,Z 650.75,A -85,B 0,C 180,E1 -20219.058,E2 -20219.058} C_VEL
LIN {X 0,Y 234.041,Z 691.719,A -85,B 0,C 180,E1 -20221.16,E2 -20221.16} C_VEL
LIN {X 0,Y 231.597,Z 744.884,A -85,B 0,C 180,E1 -20223.165,E2 -20223.165} C_VEL
LIN {X 0,Y 230.528,Z 758.311,A -85,B 0,C 180,E1 -20224.006,E2 -20224.006} C_VEL
LIN {X 0,Y 229.084,Z 770.128,A -85,B 0,C 180,E1 -20225.048,E2 -20225.048} C_VEL
LIN {X 0,Y 227.284,Z 782.6,A -85,B 0,C 180,E1 -20226.538,E2 -20226.538} C_VEL
LIN {X 0,Y 225.556,Z 793.882,A -85,B 0,C 180,E1 -20228.282,E2 -20228.282} C_VEL
LIN {X 0,Y 224.007,Z 803.518,A -85,B 0,C 180,E1 -20230.146,E2 -20230.146} C_VEL
LIN {X 0,Y 222.294,Z 813.341,A -85,B 0,C 180,E1 -20232.519,E2 -20232.519} C_VEL
LIN {X 0,Y 220.837,Z 822.352,A -85,B 0,C 180,E1 -20235.248,E2 -20235.248} C_VEL
LIN {X 0,Y 219.73,Z 829.495,A -85,B 0,C 180,E1 -20237.999,E2 -20237.999} C_VEL
LIN {X 0,Y 219.192,Z 835.186,A -85,B 0,C 180,E1 -20240.773,E2 -20240.773} C_VEL
LIN {X 0,Y 218.958,Z 839.718,A -85,B 0,C 180,E1 -20243.64,E2 -20243.64} C_VEL
LIN {X 0,Y 218.936,Z 842.834,A -85,B 0,C 180,E1 -20246.317,E2 -20246.317} C_VEL
LIN {X 0,Y 218.894,Z 844.394,A -85,B 0,C 180,E1 -20248.158,E2 -20248.158} C_VEL
LIN {X 0,Y 218.946,Z 845.517,A -85,B 0,C 180,E1 -20249.998,E2 -20249.998} C_VEL
LIN {X 0,Y 218.843,Z 846.15,A -85,B 0,C 180,E1 -20251.838,E2 -20251.838} C_VEL
LIN {X 0,Y 218.708,Z 846.27,A -85,B 0,C 180,E1 -20255.019,E2 -20255.019} C_VEL
LIN {X 0,Y 218.777,Z 845.599,A -85,B 0,C 180,E1 -20257.381,E2 -20257.381} C_VEL
LIN {X 0,Y 219.467,Z 843.165,A -85,B 0,C 180,E1 -20261.075,E2 -20261.075} C_VEL
LIN {X 0,Y 220.502,Z 840.261,A -85,B 0,C 180,E1 -20263.828,E2 -20263.828} C_VEL
LIN {X 0,Y 222.193,Z 836.348,A -85,B 0,C 180,E1 -20266.537,E2 -20266.537} C_VEL
LIN {X 0,Y 224.253,Z 831.376,A -85,B 0,C 180,E1 -20269.21,E2 -20269.21} C_VEL
LIN {X 0,Y 227.299,Z 824.031,A -85,B 0,C 180,E1 -20272.255,E2 -20272.255} C_VEL
LIN {X 0,Y 230.516,Z 816.15,A -85,B 0,C 180,E1 -20274.783,E2 -20274.783} C_VEL
LIN {X 0,Y 234.283,Z 806.381,A -85,B 0,C 180,E1 -20277.222,E2 -20277.222} C_VEL
LIN {X 0,Y 237.827,Z 796.504,A -85,B 0,C 180,E1 -20279.18,E2 -20279.18} C_VEL
LIN {X 0,Y 241.363,Z 785.567,A -85,B 0,C 180,E1 -20280.875,E2 -20280.875} C_VEL
LIN {X 0,Y 244.788,Z 773.386,A -85,B 0,C 180,E1 -20282.324,E2 -20282.324} C_VEL
LIN {X 0,Y 247.462,Z 761.792,A -85,B 0,C 180,E1 -20283.382,E2 -20283.382} C_VEL
LIN {X 0,Y 249.827,Z 748.334,A -85,B 0,C 180,E1 -20284.279,E2 -20284.279} C_VEL
LIN {X 0,Y 251.519,Z 734.494,A -85,B 0,C 180,E1 -20284.889,E2 -20284.889} C_VEL
LIN {X 0,Y 254.618,Z 696.155,A -85,B 0,C 180,E1 -20286.268,E2 -20286.268} C_VEL
LIN {X 0,Y 253.752,Z 682.394,A -85,B 0,C 180,E1 -20287.297,E2 -20287.297} C_VEL
LIN {X 0,Y 253.21,Z 677.919,A -85,B 0,C 180,E1 -20287.714,E2 -20287.714} C_VEL
LIN {X 0,Y 248.858,Z 667.284,A -85,B 0,C 180,E1 -20289.698,E2 -20289.698} C_VEL
LIN {X 0,Y 244.462,Z 658.195,A -85,B 0,C 180,E1 -20291.844,E2 -20291.844} C_VEL
LIN {X 0,Y 240.942,Z 651.835,A -85,B 0,C 180,E1 -20293.718,E2 -20293.718} C_VEL
LIN {X 0,Y 237.816,Z 646.379,A -85,B 0,C 180,E1 -20295.607,E2 -20295.607} C_VEL
LIN {X 0,Y 234.51,Z 640.991,A -85,B 0,C 180,E1 -20297.856,E2 -20297.856} C_VEL
LIN {X 0,Y 232.335,Z 638.048,A -85,B 0,C 180,E1 -20299.511,E2 -20299.511} C_VEL
LIN {X 0,Y 229.127,Z 632.731,A -85,B 0,C 180,E1 -20302.672,E2 -20302.672} C_VEL
LIN {X 0,Y 225.912,Z 628.573,A -85,B 0,C 180,E1 -20307.229,E2 -20307.229} C_VEL
LIN {X 0,Y 224.666,Z 626.391,A -85,B 0,C 180,E1 -20311.455,E2 -20311.455} C_VEL
LIN {X 0,Y 224.845,Z 625.783,A -85,B 0,C 180,E1 -20315.015,E2 -20315.015} C_VEL
LIN {X 0,Y 226.653,Z 626.921,A -85,B 0,C 180,E1 -20319.536,E2 -20319.536} C_VEL
LIN {X 0,Y 227.837,Z 627.783,A -85,B 0,C 180,E1 -20321.218,E2 -20321.218} C_VEL
LIN {X 0,Y 231.872,Z 631.991,A -85,B 0,C 180,E1 -20325.474,E2 -20325.474} C_VEL
LIN {X 0,Y 232.643,Z 632.865,A -85,B 0,C 180,E1 -20326.126,E2 -20326.126} C_VEL
LIN {X 0,Y 235.627,Z 636.471,A -85,B 0,C 180,E1 -20328.36,E2 -20328.36} C_VEL
LIN {X 0,Y 236.927,Z 637.76,A -85,B 0,C 180,E1 -20329.207,E2 -20329.207} C_VEL
LIN {X 0,Y 240.384,Z 642.474,A -85,B 0,C 180,E1 -20331.303,E2 -20331.303} C_VEL
LIN {X 0,Y 246.257,Z 650.857,A -85,B 0,C 180,E1 -20334.338,E2 -20334.338} C_VEL
LIN {X 0,Y 249.718,Z 656.484,A -85,B 0,C 180,E1 -20335.913,E2 -20335.913} C_VEL
LIN {X 0,Y 256.265,Z 669.76,A -85,B 0,C 180,E1 -20338.694,E2 -20338.694} C_VEL
LIN {X 0,Y 256.414,Z 670.668,A -85,B 0,C 180,E1 -20338.788,E2 -20338.788} C_VEL
LIN {X 0,Y 252.086,Z 721.167,A -85,B 0,C 180,E1 -20340.598,E2 -20340.598} C_VEL
LIN {X 0,Y 250.507,Z 733.698,A -85,B 0,C 180,E1 -20341.306,E2 -20341.306} C_VEL
LIN {X 0,Y 248.262,Z 747.197,A -85,B 0,C 180,E1 -20342.421,E2 -20342.421} C_VEL
LIN {X 0,Y 245.699,Z 758.534,A -85,B 0,C 180,E1 -20343.648,E2 -20343.648} C_VEL
LIN {X 0,Y 242.397,Z 770.609,A -85,B 0,C 180,E1 -20345.361,E2 -20345.361} C_VEL
LIN {X 0,Y 239.241,Z 780.564,A -85,B 0,C 180,E1 -20347.172,E2 -20347.172} C_VEL
LIN {X 0,Y 235.554,Z 790.267,A -85,B 0,C 180,E1 -20349.391,E2 -20349.391} C_VEL
LIN {X 0,Y 232.169,Z 798.503,A -85,B 0,C 180,E1 -20351.79,E2 -20351.79} C_VEL
LIN {X 0,Y 229.2,Z 805.057,A -85,B 0,C 180,E1 -20354.2,E2 -20354.2} C_VEL
LIN {X 0,Y 226.162,Z 811.223,A -85,B 0,C 180,E1 -20357.169,E2 -20357.169} C_VEL
LIN {X 0,Y 223.748,Z 815.864,A -85,B 0,C 180,E1 -20360.213,E2 -20360.213} C_VEL
LIN {X 0,Y 221.862,Z 819.132,A -85,B 0,C 180,E1 -20363.277,E2 -20363.277} C_VEL
LIN {X 0,Y 220.269,Z 821.285,A -85,B 0,C 180,E1 -20366.704,E2 -20366.704} C_VEL
LIN {X 0,Y 219.251,Z 821.984,A -85,B 0,C 180,E1 -20370.068,E2 -20370.068} C_VEL
LIN {X 0,Y 218.709,Z 821.377,A -85,B 0,C 180,E1 -20373.338,E2 -20373.338} C_VEL
LIN {X 0,Y 218.599,Z 819.558,A -85,B 0,C 180,E1 -20376.514,E2 -20376.514} C_VEL
LIN {X 0,Y 218.886,Z 816.116,A -85,B 0,C 180,E1 -20379.953,E2 -20379.953} C_VEL
LIN {X 0,Y 219.382,Z 812.465,A -85,B 0,C 180,E1 -20382.543,E2 -20382.543} C_VEL
LIN {X 0,Y 220.129,Z 807.251,A -85,B 0,C 180,E1 -20385.384,E2 -20385.384} C_VEL
LIN {X 0,Y 221.132,Z 800.837,A -85,B 0,C 180,E1 -20388.135,E2 -20388.135} C_VEL
LIN {X 0,Y 222.493,Z 792.98,A -85,B 0,C 180,E1 -20390.823,E2 -20390.823} C_VEL
LIN {X 0,Y 224.184,Z 783.286,A -85,B 0,C 180,E1 -20393.445,E2 -20393.445} C_VEL
LIN {X 0,Y 225.837,Z 773.582,A -85,B 0,C 180,E1 -20395.555,E2 -20395.555} C_VEL
LIN {X 0,Y 227.472,Z 763.396,A -85,B 0,C 180,E1 -20397.343,E2 -20397.343} C_VEL
LIN {X 0,Y 229.096,Z 750.944,A -85,B 0,C 180,E1 -20399.07,E2 -20399.07} C_VEL
LIN {X 0,Y 230.461,Z 739.427,A -85,B 0,C 180,E1 -20400.296,E2 -20400.296} C_VEL
LIN {X 0,Y 231.555,Z 725.959,A -85,B 0,C 180,E1 -20401.354,E2 -20401.354} C_VEL
LIN {X 0,Y 232.384,Z 712.157,A -85,B 0,C 180,E1 -20402.06,E2 -20402.06} C_VEL
LIN {X 0,Y 235.007,Z 652.549,A -85,B 0,C 180,E1 -20404.245,E2 -20404.245} C_VEL
LIN {X 0,Y 224.435,Z 626.474,A -85,B 0,C 180,E1 -20406.399,E2 -20406.399} C_VEL
LIN {X 0,Y 221.048,Z 618.758,A -85,B 0,C 180,E1 -20407.104,E2 -20407.104} C_VEL
LIN {X 0,Y 220.908,Z 617.968,A -85,B 0,C 180,E1 -20407.187,E2 -20407.187} C_VEL
LIN {X 0,Y 220.926,Z 617.964,A -85,B 0,C 180,E1 -20411.453,E2 -20411.453} C_VEL
LIN {X 0,Y 220.996,Z 617.955,A -85,B 0,C 180,E1 -20415.263,E2 -20415.263} C_VEL
LIN {X 0,Y 221.258,Z 617.925,A -85,B 0,C 180,E1 -20420.864,E2 -20420.864} C_VEL
LIN {X 0,Y 221.311,Z 617.919,A -85,B 0,C 180,E1 -20422.704,E2 -20422.704} C_VEL
LIN {X 0,Y 221.514,Z 617.893,A -85,B 0,C 180,E1 -20428.184,E2 -20428.184} C_VEL
LIN {X 0,Y 221.517,Z 617.89,A -85,B 0,C 180,E1 -20431.82,E2 -20431.82} C_VEL
LIN {X 0,Y 221.313,Z 617.915,A -85,B 0,C 180,E1 -20437.3,E2 -20437.3} C_VEL
LIN {X 0,Y 221.119,Z 617.94,A -85,B 0,C 180,E1 -20440.996,E2 -20440.996} C_VEL
LIN {X 0,Y 221.019,Z 617.953,A -85,B 0,C 180,E1 -20446.632,E2 -20446.632} C_VEL
LIN {X 0,Y 220.896,Z 617.957,A -85,B 0,C 180,E1 -20450.488,E2 -20450.488} C_VEL
LIN {X 0,Y 220.871,Z 617.97,A -85,B 0,C 180,E1 -20454.437,E2 -20454.437} C_VEL
LIN {X 0,Y 220.84,Z 617.974,A -85,B 0,C 180,E1 -20458.515,E2 -20458.515} C_VEL
LIN {X 0,Y 220.821,Z 617.966,A -85,B 0,C 180,E1 -20462.757,E2 -20462.757} C_VEL
LIN {X 0,Y 220.814,Z 617.971,A -85,B 0,C 180,E1 -20467.28,E2 -20467.28} C_VEL
LIN {X 0,Y 220.775,Z 617.981,A -85,B 0,C 180,E1 -20471.954,E2 -20471.954} C_VEL
LIN {X 0,Y 220.78,Z 617.979,A -85,B 0,C 180,E1 -20475.548,E2 -20475.548} C_VEL
LIN {X 0,Y 220.812,Z 617.961,A -85,B 0,C 180,E1 -20480.464,E2 -20480.464} C_VEL
LIN {X 0,Y 220.809,Z 617.963,A -85,B 0,C 180,E1 -20485.047,E2 -20485.047} C_VEL
LIN {X 0,Y 220.874,Z 617.968,A -85,B 0,C 180,E1 -20489.396,E2 -20489.396} C_VEL
LIN {X 0,Y 220.901,Z 617.97,A -85,B 0,C 180,E1 -20493.55,E2 -20493.55} C_VEL
LIN {X 0,Y 220.872,Z 617.969,A -85,B 0,C 180,E1 -20497.553,E2 -20497.553} C_VEL
LIN {X 0,Y 220.99,Z 617.934,A -85,B 0,C 180,E1 -20502.573,E2 -20502.573} C_VEL
LIN {X 0,Y 221.016,Z 617.942,A -85,B 0,C 180,E1 -20507.139,E2 -20507.139} C_VEL
LIN {X 0,Y 221.212,Z 617.926,A -85,B 0,C 180,E1 -20510.86,E2 -20510.86} C_VEL
LIN {X 0,Y 221.266,Z 617.921,A -85,B 0,C 180,E1 -20512.701,E2 -20512.701} C_VEL
LIN {X 0,Y 221.519,Z 617.885,A -85,B 0,C 180,E1 -20518.182,E2 -20518.182} C_VEL
LIN {X 0,Y 221.519,Z 617.875,A -85,B 0,C 180,E1 -20521.818,E2 -20521.818} C_VEL
LIN {X 0,Y 221.267,Z 617.92,A -85,B 0,C 180,E1 -20527.299,E2 -20527.299} C_VEL
LIN {X 0,Y 221.073,Z 617.945,A -85,B 0,C 180,E1 -20530.996,E2 -20530.996} C_VEL
LIN {X 0,Y 220.976,Z 617.95,A -85,B 0,C 180,E1 -20534.74,E2 -20534.74} C_VEL
LIN {X 0,Y 220.895,Z 617.97,A -85,B 0,C 180,E1 -20538.552,E2 -20538.552} C_VEL
LIN {X 0,Y 220.891,Z 617.971,A -85,B 0,C 180,E1 -20542.674,E2 -20542.674} C_VEL
LIN {X 0,Y 220.893,Z 617.97,A -85,B 0,C 180,E1 -20547.015,E2 -20547.015} C_VEL
LIN {X 0,Y 220.87,Z 617.974,A -85,B 0,C 180,E1 -20550.778,E2 -20550.778} C_VEL
LIN {X 0,Y 220.785,Z 617.981,A -85,B 0,C 180,E1 -20555.41,E2 -20555.41} C_VEL
LIN {X 0,Y 220.813,Z 617.98,A -85,B 0,C 180,E1 -20559.536,E2 -20559.536} C_VEL
LIN {X 0,Y 220.761,Z 617.988,A -85,B 0,C 180,E1 -20563.315,E2 -20563.315} C_VEL
LIN {X 0,Y 220.061,Z 618.075,A -85,B 0,C 180,E1 -20564.327,E2 -20564.327} C_VEL
LIN {X 0,Y 217.182,Z 618.432,A -85,B 0,C 180,E1 -20565.916,E2 -20565.916} C_VEL
LIN {X 0,Y 214.325,Z 618.789,A -85,B 0,C 180,E1 -20567.546,E2 -20567.546} C_VEL
LIN {X 0,Y 213.698,Z 618.865,A -85,B 0,C 180,E1 -20568.604,E2 -20568.604} C_VEL
LIN {X 0,Y 213.779,Z 618.904,A -85,B 0,C 180,E1 -20570.383,E2 -20570.383} C_VEL
LIN {X 0,Y 215.866,Z 628.432,A -85,B 0,C 180,E1 -20574.483,E2 -20574.483} C_VEL
LIN {X 0,Y 217.195,Z 634.75,A -85,B 0,C 180,E1 -20577.064,E2 -20577.064} C_VEL
LIN {X 0,Y 223.064,Z 652.651,A -85,B 0,C 180,E1 -20578.492,E2 -20578.492} C_VEL
LIN {X 0,Y 227.318,Z 692.849,A -85,B 0,C 180,E1 -20580.621,E2 -20580.621} C_VEL
LIN {X 0,Y 224.883,Z 744.098,A -85,B 0,C 180,E1 -20582.612,E2 -20582.612} C_VEL
LIN {X 0,Y 223.795,Z 757.625,A -85,B 0,C 180,E1 -20583.477,E2 -20583.477} C_VEL
LIN {X 0,Y 222.227,Z 770.018,A -85,B 0,C 180,E1 -20584.599,E2 -20584.599} C_VEL
LIN {X 0,Y 220.517,Z 781.637,A -85,B 0,C 180,E1 -20586.022,E2 -20586.022} C_VEL
LIN {X 0,Y 218.729,Z 793.016,A -85,B 0,C 180,E1 -20587.817,E2 -20587.817} C_VEL
LIN {X 0,Y 217.198,Z 802.098,A -85,B 0,C 180,E1 -20589.6,E2 -20589.6} C_VEL
LIN {X 0,Y 215.465,Z 811.804,A -85,B 0,C 180,E1 -20591.947,E2 -20591.947} C_VEL
LIN {X 0,Y 213.948,Z 821.01,A -85,B 0,C 180,E1 -20594.762,E2 -20594.762} C_VEL
LIN {X 0,Y 212.755,Z 828.376,A -85,B 0,C 180,E1 -20597.599,E2 -20597.599} C_VEL
LIN {X 0,Y 212.154,Z 834.218,A -85,B 0,C 180,E1 -20600.464,E2 -20600.464} C_VEL
LIN {X 0,Y 211.894,Z 838.753,A -85,B 0,C 180,E1 -20603.332,E2 -20603.332} C_VEL
LIN {X 0,Y 211.877,Z 842.116,A -85,B 0,C 180,E1 -20606.194,E2 -20606.194} C_VEL
LIN {X 0,Y 211.827,Z 843.726,A -85,B 0,C 180,E1 -20608.097,E2 -20608.097} C_VEL
LIN {X 0,Y 211.872,Z 844.907,A -85,B 0,C 180,E1 -20609.998,E2 -20609.998} C_VEL
LIN {X 0,Y 211.771,Z 845.637,A -85,B 0,C 180,E1 -20611.9,E2 -20611.9} C_VEL
LIN {X 0,Y 211.623,Z 845.906,A -85,B 0,C 180,E1 -20614.924,E2 -20614.924} C_VEL
LIN {X 0,Y 211.7,Z 845.257,A -85,B 0,C 180,E1 -20617.629,E2 -20617.629} C_VEL
LIN {X 0,Y 212.005,Z 844.344,A -85,B 0,C 180,E1 -20619.539,E2 -20619.539} C_VEL
LIN {X 0,Y 213.121,Z 841.232,A -85,B 0,C 180,E1 -20623.344,E2 -20623.344} C_VEL
LIN {X 0,Y 214.735,Z 837.814,A -85,B 0,C 180,E1 -20626.15,E2 -20626.15} C_VEL
LIN {X 0,Y 216.777,Z 833.354,A -85,B 0,C 180,E1 -20628.915,E2 -20628.915} C_VEL
LIN {X 0,Y 219.485,Z 827.362,A -85,B 0,C 180,E1 -20631.783,E2 -20631.783} C_VEL
LIN {X 0,Y 222.946,Z 819.562,A -85,B 0,C 180,E1 -20634.686,E2 -20634.686} C_VEL
LIN {X 0,Y 226.733,Z 810.773,A -85,B 0,C 180,E1 -20637.204,E2 -20637.204} C_VEL
LIN {X 0,Y 230.204,Z 801.898,A -85,B 0,C 180,E1 -20639.238,E2 -20639.238} C_VEL
LIN {X 0,Y 234.111,Z 791.103,A -85,B 0,C 180,E1 -20641.185,E2 -20641.185} C_VEL
LIN {X 0,Y 238.013,Z 778.885,A -85,B 0,C 180,E1 -20642.856,E2 -20642.856} C_VEL
LIN {X 0,Y 241.18,Z 767.02,A -85,B 0,C 180,E1 -20644.119,E2 -20644.119} C_VEL
LIN {X 0,Y 243.854,Z 754.903,A -85,B 0,C 180,E1 -20645.07,E2 -20645.07} C_VEL
LIN {X 0,Y 246.008,Z 741.514,A -85,B 0,C 180,E1 -20645.814,E2 -20645.814} C_VEL
LIN {X 0,Y 249.047,Z 708.122,A -85,B 0,C 180,E1 -20647.06,E2 -20647.06} C_VEL
LIN {X 0,Y 249.928,Z 696.722,A -85,B 0,C 180,E1 -20647.502,E2 -20647.502} C_VEL
LIN {X 0,Y 249.243,Z 684.443,A -85,B 0,C 180,E1 -20648.457,E2 -20648.457} C_VEL
LIN {X 0,Y 248.893,Z 681.492,A -85,B 0,C 180,E1 -20648.754,E2 -20648.754} C_VEL
LIN {X 0,Y 245.07,Z 671.837,A -85,B 0,C 180,E1 -20650.636,E2 -20650.636} C_VEL
LIN {X 0,Y 241.28,Z 663.526,A -85,B 0,C 180,E1 -20652.656,E2 -20652.656} C_VEL
LIN {X 0,Y 237.996,Z 657.375,A -85,B 0,C 180,E1 -20654.537,E2 -20654.537} C_VEL
LIN {X 0,Y 235.153,Z 652.222,A -85,B 0,C 180,E1 -20656.375,E2 -20656.375} C_VEL
LIN {X 0,Y 231.709,Z 646.259,A -85,B 0,C 180,E1 -20658.961,E2 -20658.961} C_VEL
LIN {X 0,Y 227.312,Z 639.265,A -85,B 0,C 180,E1 -20663.246,E2 -20663.246} C_VEL
LIN {X 0,Y 224.455,Z 635.308,A -85,B 0,C 180,E1 -20667.711,E2 -20667.711} C_VEL
LIN {X 0,Y 223.413,Z 633.291,A -85,B 0,C 180,E1 -20671.844,E2 -20671.844} C_VEL
LIN {X 0,Y 223.452,Z 632.814,A -85,B 0,C 180,E1 -20673.875,E2 -20673.875} C_VEL
LIN {X 0,Y 224.586,Z 633.316,A -85,B 0,C 180,E1 -20677.943,E2 -20677.943} C_VEL
LIN {X 0,Y 226.405,Z 634.708,A -85,B 0,C 180,E1 -20680.977,E2 -20680.977} C_VEL
LIN {X 0,Y 230.284,Z 638.832,A -85,B 0,C 180,E1 -20685.209,E2 -20685.209} C_VEL
LIN {X 0,Y 233.759,Z 643.15,A -85,B 0,C 180,E1 -20687.991,E2 -20687.991} C_VEL
LIN {X 0,Y 234.89,Z 644.403,A -85,B 0,C 180,E1 -20688.776,E2 -20688.776} C_VEL
LIN {X 0,Y 237.982,Z 648.786,A -85,B 0,C 180,E1 -20690.752,E2 -20690.752} C_VEL
LIN {X 0,Y 243.102,Z 656.274,A -85,B 0,C 180,E1 -20693.554,E2 -20693.554} C_VEL
LIN {X 0,Y 246.515,Z 662.197,A -85,B 0,C 180,E1 -20695.247,E2 -20695.247} C_VEL
LIN {X 0,Y 251.642,Z 672.933,A -85,B 0,C 180,E1 -20697.593,E2 -20697.593} C_VEL
LIN {X 0,Y 247.282,Z 722.726,A -85,B 0,C 180,E1 -20699.45,E2 -20699.45} C_VEL
LIN {X 0,Y 245.572,Z 735.088,A -85,B 0,C 180,E1 -20700.166,E2 -20700.166} C_VEL
LIN {X 0,Y 243.375,Z 747.385,A -85,B 0,C 180,E1 -20701.199,E2 -20701.199} C_VEL
LIN {X 0,Y 240.821,Z 758.256,A -85,B 0,C 180,E1 -20702.382,E2 -20702.382} C_VEL
LIN {X 0,Y 237.494,Z 769.881,A -85,B 0,C 180,E1 -20704.03,E2 -20704.03} C_VEL
LIN {X 0,Y 234.359,Z 779.359,A -85,B 0,C 180,E1 -20705.718,E2 -20705.718} C_VEL
LIN {X 0,Y 230.602,Z 789.128,A -85,B 0,C 180,E1 -20707.882,E2 -20707.882} C_VEL
LIN {X 0,Y 227.329,Z 796.687,A -85,B 0,C 180,E1 -20710.003,E2 -20710.003} C_VEL
LIN {X 0,Y 223.498,Z 804.73,A -85,B 0,C 180,E1 -20712.898,E2 -20712.898} C_VEL
LIN {X 0,Y 220.535,Z 810.378,A -85,B 0,C 180,E1 -20715.53,E2 -20715.53} C_VEL
LIN {X 0,Y 217.639,Z 815.634,A -85,B 0,C 180,E1 -20718.839,E2 -20718.839} C_VEL
LIN {X 0,Y 216.118,Z 818.132,A -85,B 0,C 180,E1 -20720.96,E2 -20720.96} C_VEL
LIN {X 0,Y 214.601,Z 820.328,A -85,B 0,C 180,E1 -20723.518,E2 -20723.518} C_VEL
LIN {X 0,Y 213.046,Z 822.084,A -85,B 0,C 180,E1 -20727.046,E2 -20727.046} C_VEL
LIN {X 0,Y 212.056,Z 822.406,A -85,B 0,C 180,E1 -20730.497,E2 -20730.497} C_VEL
LIN {X 0,Y 211.577,Z 821.424,A -85,B 0,C 180,E1 -20733.861,E2 -20733.861} C_VEL
LIN {X 0,Y 211.516,Z 819.259,A -85,B 0,C 180,E1 -20737.117,E2 -20737.117} C_VEL
LIN {X 0,Y 211.848,Z 815.958,A -85,B 0,C 180,E1 -20740.272,E2 -20740.272} C_VEL
LIN {X 0,Y 212.445,Z 811.56,A -85,B 0,C 180,E1 -20743.302,E2 -20743.302} C_VEL
LIN {X 0,Y 213.366,Z 805.523,A -85,B 0,C 180,E1 -20746.44,E2 -20746.44} C_VEL
LIN {X 0,Y 214.678,Z 797.768,A -85,B 0,C 180,E1 -20749.564,E2 -20749.564} C_VEL
LIN {X 0,Y 216.175,Z 789.364,A -85,B 0,C 180,E1 -20752.237,E2 -20752.237} C_VEL
LIN {X 0,Y 218.045,Z 778.885,A -85,B 0,C 180,E1 -20754.872,E2 -20754.872} C_VEL
LIN {X 0,Y 219.911,Z 767.693,A -85,B 0,C 180,E1 -20757.095,E2 -20757.095} C_VEL
LIN {X 0,Y 221.616,Z 756.162,A -85,B 0,C 180,E1 -20758.896,E2 -20758.896} C_VEL
LIN {X 0,Y 223.2,Z 743.982,A -85,B 0,C 180,E1 -20760.377,E2 -20760.377} C_VEL
LIN {X 0,Y 224.526,Z 730.401,A -85,B 0,C 180,E1 -20761.589,E2 -20761.589} C_VEL
LIN {X 0,Y 225.405,Z 717.3,A -85,B 0,C 180,E1 -20762.401,E2 -20762.401} C_VEL
LIN {X 0,Y 228.358,Z 654.199,A -85,B 0,C 180,E1 -20764.806,E2 -20764.806} C_VEL
LIN {X 0,Y 218.411,Z 629.682,A -85,B 0,C 180,E1 -20766.908,E2 -20766.908} C_VEL
LIN {X 0,Y 213.986,Z 619.454,A -85,B 0,C 180,E1 -20767.875,E2 -20767.875} C_VEL
LIN {X 0,Y 213.885,Z 618.842,A -85,B 0,C 180,E1 -20767.927,E2 -20767.927} C_VEL
LIN {X 0,Y 213.943,Z 618.834,A -85,B 0,C 180,E1 -20772.806,E2 -20772.806} C_VEL
LIN {X 0,Y 213.98,Z 618.83,A -85,B 0,C 180,E1 -20776.71,E2 -20776.71} C_VEL
LIN {X 0,Y 214.196,Z 618.806,A -85,B 0,C 180,E1 -20780.56,E2 -20780.56} C_VEL
LIN {X 0,Y 214.248,Z 618.799,A -85,B 0,C 180,E1 -20782.462,E2 -20782.462} C_VEL
LIN {X 0,Y 214.448,Z 618.773,A -85,B 0,C 180,E1 -20788.124,E2 -20788.124} C_VEL
LIN {X 0,Y 214.551,Z 618.759,A -85,B 0,C 180,E1 -20790.002,E2 -20790.002} C_VEL
LIN {X 0,Y 214.45,Z 618.771,A -85,B 0,C 180,E1 -20791.88,E2 -20791.88} C_VEL
LIN {X 0,Y 214.25,Z 618.794,A -85,B 0,C 180,E1 -20797.542,E2 -20797.542} C_VEL
LIN {X 0,Y 214.05,Z 618.819,A -85,B 0,C 180,E1 -20801.364,E2 -20801.364} C_VEL
LIN {X 0,Y 213.937,Z 618.834,A -85,B 0,C 180,E1 -20805.239,E2 -20805.239} C_VEL
LIN {X 0,Y 213.842,Z 618.835,A -85,B 0,C 180,E1 -20809.189,E2 -20809.189} C_VEL
LIN {X 0,Y 213.851,Z 618.846,A -85,B 0,C 180,E1 -20813.229,E2 -20813.229} C_VEL
LIN {X 0,Y 213.833,Z 618.847,A -85,B 0,C 180,E1 -20817.451,E2 -20817.451} C_VEL
LIN {X 0,Y 213.781,Z 618.843,A -85,B 0,C 180,E1 -20821.738,E2 -20821.738} C_VEL
LIN {X 0,Y 213.748,Z 618.846,A -85,B 0,C 180,E1 -20826.29,E2 -20826.29} C_VEL
LIN {X 0,Y 213.717,Z 618.862,A -85,B 0,C 180,E1 -20831.126,E2 -20831.126} C_VEL
LIN {X 0,Y 213.712,Z 618.862,A -85,B 0,C 180,E1 -20833.679,E2 -20833.679} C_VEL
LIN {X 0,Y 213.712,Z 618.857,A -85,B 0,C 180,E1 -20836.345,E2 -20836.345} C_VEL
LIN {X 0,Y 213.722,Z 618.85,A -85,B 0,C 180,E1 -20839.144,E2 -20839.144} C_VEL
LIN {X 0,Y 213.75,Z 618.836,A -85,B 0,C 180,E1 -20843.713,E2 -20843.713} C_VEL
LIN {X 0,Y 213.801,Z 618.846,A -85,B 0,C 180,E1 -20848.726,E2 -20848.726} C_VEL
LIN {X 0,Y 213.832,Z 618.847,A -85,B 0,C 180,E1 -20852.604,E2 -20852.604} C_VEL
LIN {X 0,Y 213.826,Z 618.845,A -85,B 0,C 180,E1 -20856.975,E2 -20856.975} C_VEL
LIN {X 0,Y 213.949,Z 618.81,A -85,B 0,C 180,E1 -20862.804,E2 -20862.804} C_VEL
LIN {X 0,Y 213.957,Z 618.82,A -85,B 0,C 180,E1 -20866.707,E2 -20866.707} C_VEL
LIN {X 0,Y 214.149,Z 618.806,A -85,B 0,C 180,E1 -20870.556,E2 -20870.556} C_VEL
LIN {X 0,Y 214.107,Z 618.814,A -85,B 0,C 180,E1 -20874.349,E2 -20874.349} C_VEL
LIN {X 0,Y 214.452,Z 618.765,A -85,B 0,C 180,E1 -20878.122,E2 -20878.122} C_VEL
LIN {X 0,Y 214.557,Z 618.746,A -85,B 0,C 180,E1 -20880,E2 -20880} C_VEL
LIN {X 0,Y 214.452,Z 618.755,A -85,B 0,C 180,E1 -20881.878,E2 -20881.878} C_VEL
LIN {X 0,Y 214.206,Z 618.8,A -85,B 0,C 180,E1 -20887.541,E2 -20887.541} C_VEL
LIN {X 0,Y 214.004,Z 618.825,A -85,B 0,C 180,E1 -20891.364,E2 -20891.364} C_VEL
LIN {X 0,Y 213.91,Z 618.829,A -85,B 0,C 180,E1 -20895.239,E2 -20895.239} C_VEL
LIN {X 0,Y 213.819,Z 618.851,A -85,B 0,C 180,E1 -20899.19,E2 -20899.19} C_VEL
LIN {X 0,Y 213.817,Z 618.849,A -85,B 0,C 180,E1 -20903.231,E2 -20903.231} C_VEL
LIN {X 0,Y 213.836,Z 618.848,A -85,B 0,C 180,E1 -20907.449,E2 -20907.449} C_VEL
LIN {X 0,Y 213.784,Z 618.853,A -85,B 0,C 180,E1 -20911.735,E2 -20911.735} C_VEL
LIN {X 0,Y 213.75,Z 618.858,A -85,B 0,C 180,E1 -20916.287,E2 -20916.287} C_VEL
LIN {X 0,Y 213.719,Z 618.866,A -85,B 0,C 180,E1 -20921.124,E2 -20921.124} C_VEL
LIN {X 0,Y 213.714,Z 618.865,A -85,B 0,C 180,E1 -20923.677,E2 -20923.677} C_VEL
LIN {X 0,Y 213.713,Z 618.865,A -85,B 0,C 180,E1 -20926.342,E2 -20926.342} C_VEL
LIN {X 0,Y 213.698,Z 618.865,A -85,B 0,C 180,E1 -20928.604,E2 -20928.604} C_VEL
LIN {X 0,Y 213.535,Z 619.375,A -85,B 0,C 180,E1 -20929.641,E2 -20929.641} C_VEL
LIN {X 0,Y 213.028,Z 620.672,A -85,B 0,C 180,E1 -20930.628,E2 -20930.628} C_VEL
LIN {X 0,Y 211.504,Z 624.63,A -85,B 0,C 180,E1 -20932.465,E2 -20932.465} C_VEL
LIN {X 0,Y 209.706,Z 631.675,A -85,B 0,C 180,E1 -20935.139,E2 -20935.139} C_VEL
LIN {X 0,Y 209.778,Z 633.909,A -85,B 0,C 180,E1 -20936.055,E2 -20936.055} C_VEL
LIN {X 0,Y 209.968,Z 634.765,A -85,B 0,C 180,E1 -20936.248,E2 -20936.248} C_VEL
LIN {X 0,Y 216.54,Z 653.933,A -85,B 0,C 180,E1 -20937.86,E2 -20937.86} C_VEL
LIN {X 0,Y 220.634,Z 693.336,A -85,B 0,C 180,E1 -20940.022,E2 -20940.022} C_VEL
LIN {X 0,Y 218.091,Z 744.292,A -85,B 0,C 180,E1 -20942.076,E2 -20942.076} C_VEL
LIN {X 0,Y 216.863,Z 758.308,A -85,B 0,C 180,E1 -20943.016,E2 -20943.016} C_VEL
LIN {X 0,Y 215.377,Z 769.894,A -85,B 0,C 180,E1 -20944.121,E2 -20944.121} C_VEL
LIN {X 0,Y 213.504,Z 782.237,A -85,B 0,C 180,E1 -20945.701,E2 -20945.701} C_VEL
LIN {X 0,Y 211.672,Z 793.439,A -85,B 0,C 180,E1 -20947.551,E2 -20947.551} C_VEL
LIN {X 0,Y 209.861,Z 803.882,A -85,B 0,C 180,E1 -20949.745,E2 -20949.745} C_VEL
LIN {X 0,Y 208.052,Z 813.569,A -85,B 0,C 180,E1 -20952.299,E2 -20952.299} C_VEL
LIN {X 0,Y 206.815,Z 821.017,A -85,B 0,C 180,E1 -20954.728,E2 -20954.728} C_VEL
LIN {X 0,Y 205.652,Z 828.281,A -85,B 0,C 180,E1 -20957.665,E2 -20957.665} C_VEL
LIN {X 0,Y 205.114,Z 833.182,A -85,B 0,C 180,E1 -20960.133,E2 -20960.133} C_VEL
LIN {X 0,Y 204.844,Z 837.867,A -85,B 0,C 180,E1 -20963.101,E2 -20963.101} C_VEL
LIN {X 0,Y 204.82,Z 841.353,A -85,B 0,C 180,E1 -20966.063,E2 -20966.063} C_VEL
LIN {X 0,Y 204.762,Z 843.032,A -85,B 0,C 180,E1 -20968.031,E2 -20968.031} C_VEL
LIN {X 0,Y 204.799,Z 844.273,A -85,B 0,C 180,E1 -20969.998,E2 -20969.998} C_VEL
LIN {X 0,Y 204.7,Z 845.077,A -85,B 0,C 180,E1 -20971.965,E2 -20971.965} C_VEL
LIN {X 0,Y 204.55,Z 845.454,A -85,B 0,C 180,E1 -20974.864,E2 -20974.864} C_VEL
LIN {X 0,Y 204.643,Z 844.914,A -85,B 0,C 180,E1 -20977.894,E2 -20977.894} C_VEL
LIN {X 0,Y 205.462,Z 842.831,A -85,B 0,C 180,E1 -20981.841,E2 -20981.841} C_VEL
LIN {X 0,Y 206.687,Z 840.173,A -85,B 0,C 180,E1 -20984.773,E2 -20984.773} C_VEL
LIN {X 0,Y 208.613,Z 836.539,A -85,B 0,C 180,E1 -20987.648,E2 -20987.648} C_VEL
LIN {X 0,Y 210.897,Z 831.866,A -85,B 0,C 180,E1 -20990.479,E2 -20990.479} C_VEL
LIN {X 0,Y 214.264,Z 824.967,A -85,B 0,C 180,E1 -20993.689,E2 -20993.689} C_VEL
LIN {X 0,Y 217.796,Z 817.541,A -85,B 0,C 180,E1 -20996.337,E2 -20996.337} C_VEL
LIN {X 0,Y 221.928,Z 808.421,A -85,B 0,C 180,E1 -20998.875,E2 -20998.875} C_VEL
LIN {X 0,Y 225.747,Z 799.21,A -85,B 0,C 180,E1 -21000.907,E2 -21000.907} C_VEL
LIN {X 0,Y 229.487,Z 789.168,A -85,B 0,C 180,E1 -21002.665,E2 -21002.665} C_VEL
LIN {X 0,Y 233.149,Z 778.227,A -85,B 0,C 180,E1 -21004.152,E2 -21004.152} C_VEL
LIN {X 0,Y 236.715,Z 765.348,A -85,B 0,C 180,E1 -21005.505,E2 -21005.505} C_VEL
LIN {X 0,Y 239.698,Z 751.442,A -85,B 0,C 180,E1 -21006.551,E2 -21006.551} C_VEL
LIN {X 0,Y 241.786,Z 738.233,A -85,B 0,C 180,E1 -21007.223,E2 -21007.223} C_VEL
LIN {X 0,Y 245.46,Z 697.941,A -85,B 0,C 180,E1 -21008.748,E2 -21008.748} C_VEL
LIN {X 0,Y 244.908,Z 686.221,A -85,B 0,C 180,E1 -21009.704,E2 -21009.704} C_VEL
LIN {X 0,Y 244.325,Z 683.845,A -85,B 0,C 180,E1 -21010.055,E2 -21010.055} C_VEL
LIN {X 0,Y 240.672,Z 674.557,A -85,B 0,C 180,E1 -21012.034,E2 -21012.034} C_VEL
LIN {X 0,Y 237.331,Z 667.42,A -85,B 0,C 180,E1 -21013.951,E2 -21013.951} C_VEL
LIN {X 0,Y 235.174,Z 662.945,A -85,B 0,C 180,E1 -21015.353,E2 -21015.353} C_VEL
LIN {X 0,Y 232.521,Z 657.993,A -85,B 0,C 180,E1 -21017.184,E2 -21017.184} C_VEL
LIN {X 0,Y 229.463,Z 652.436,A -85,B 0,C 180,E1 -21019.674,E2 -21019.674} C_VEL
LIN {X 0,Y 225.653,Z 645.958,A -85,B 0,C 180,E1 -21023.718,E2 -21023.718} C_VEL
LIN {X 0,Y 223.138,Z 642.219,A -85,B 0,C 180,E1 -21027.927,E2 -21027.927} C_VEL
LIN {X 0,Y 222.17,Z 640.129,A -85,B 0,C 180,E1 -21032.337,E2 -21032.337} C_VEL
LIN {X 0,Y 222.571,Z 639.866,A -85,B 0,C 180,E1 -21035.764,E2 -21035.764} C_VEL
LIN {X 0,Y 224.441,Z 641.059,A -85,B 0,C 180,E1 -21039.944,E2 -21039.944} C_VEL
LIN {X 0,Y 225.913,Z 642.949,A -85,B 0,C 180,E1 -21042.052,E2 -21042.052} C_VEL
LIN {X 0,Y 228.962,Z 646.118,A -85,B 0,C 180,E1 -21045.203,E2 -21045.203} C_VEL
LIN {X 0,Y 231.754,Z 649.688,A -85,B 0,C 180,E1 -21047.522,E2 -21047.522} C_VEL
LIN {X 0,Y 232.853,Z 651.044,A -85,B 0,C 180,E1 -21048.327,E2 -21048.327} C_VEL
LIN {X 0,Y 235.636,Z 655.144,A -85,B 0,C 180,E1 -21050.213,E2 -21050.213} C_VEL
LIN {X 0,Y 240.398,Z 662.411,A -85,B 0,C 180,E1 -21052.974,E2 -21052.974} C_VEL
LIN {X 0,Y 243.561,Z 668.209,A -85,B 0,C 180,E1 -21054.634,E2 -21054.634} C_VEL
LIN {X 0,Y 247.194,Z 676.196,A -85,B 0,C 180,E1 -21056.423,E2 -21056.423} C_VEL
LIN {X 0,Y 242.747,Z 722.771,A -85,B 0,C 180,E1 -21058.156,E2 -21058.156} C_VEL
LIN {X 0,Y 240.764,Z 736.453,A -85,B 0,C 180,E1 -21058.979,E2 -21058.979} C_VEL
LIN {X 0,Y 238.275,Z 749.354,A -85,B 0,C 180,E1 -21060.105,E2 -21060.105} C_VEL
LIN {X 0,Y 235.149,Z 761.447,A -85,B 0,C 180,E1 -21061.498,E2 -21061.498} C_VEL
LIN {X 0,Y 231.63,Z 772.774,A -85,B 0,C 180,E1 -21063.198,E2 -21063.198} C_VEL
LIN {X 0,Y 228.052,Z 782.548,A -85,B 0,C 180,E1 -21065.083,E2 -21065.083} C_VEL
LIN {X 0,Y 224.286,Z 791.377,A -85,B 0,C 180,E1 -21067.2,E2 -21067.2} C_VEL
LIN {X 0,Y 220.486,Z 799.488,A -85,B 0,C 180,E1 -21069.651,E2 -21069.651} C_VEL
LIN {X 0,Y 217.34,Z 805.613,A -85,B 0,C 180,E1 -21071.998,E2 -21071.998} C_VEL
LIN {X 0,Y 214.728,Z 810.25,A -85,B 0,C 180,E1 -21074.21,E2 -21074.21} C_VEL
LIN {X 0,Y 211.68,Z 815.388,A -85,B 0,C 180,E1 -21077.386,E2 -21077.386} C_VEL
LIN {X 0,Y 209.55,Z 818.59,A -85,B 0,C 180,E1 -21080.11,E2 -21080.11} C_VEL
LIN {X 0,Y 207.358,Z 821.444,A -85,B 0,C 180,E1 -21083.784,E2 -21083.784} C_VEL
LIN {X 0,Y 205.813,Z 822.755,A -85,B 0,C 180,E1 -21087.403,E2 -21087.403} C_VEL
LIN {X 0,Y 204.852,Z 822.709,A -85,B 0,C 180,E1 -21090.971,E2 -21090.971} C_VEL
LIN {X 0,Y 204.457,Z 821.404,A -85,B 0,C 180,E1 -21094.418,E2 -21094.418} C_VEL
LIN {X 0,Y 204.503,Z 818.451,A -85,B 0,C 180,E1 -21098.213,E2 -21098.213} C_VEL
LIN {X 0,Y 205.089,Z 813.85,A -85,B 0,C 180,E1 -21102.023,E2 -21102.023} C_VEL
LIN {X 0,Y 205.756,Z 809.159,A -85,B 0,C 180,E1 -21104.864,E2 -21104.864} C_VEL
LIN {X 0,Y 206.668,Z 803.342,A -85,B 0,C 180,E1 -21107.657,E2 -21107.657} C_VEL
LIN {X 0,Y 207.935,Z 796.233,A -85,B 0,C 180,E1 -21110.4,E2 -21110.4} C_VEL
LIN {X 0,Y 209.544,Z 787.526,A -85,B 0,C 180,E1 -21113.107,E2 -21113.107} C_VEL
LIN {X 0,Y 211.347,Z 777.612,A -85,B 0,C 180,E1 -21115.579,E2 -21115.579} C_VEL
LIN {X 0,Y 213.285,Z 766.29,A -85,B 0,C 180,E1 -21117.809,E2 -21117.809} C_VEL
LIN {X 0,Y 214.957,Z 754.987,A -85,B 0,C 180,E1 -21119.578,E2 -21119.578} C_VEL
LIN {X 0,Y 216.671,Z 741.858,A -85,B 0,C 180,E1 -21121.137,E2 -21121.137} C_VEL
LIN {X 0,Y 217.92,Z 728.392,A -85,B 0,C 180,E1 -21122.318,E2 -21122.318} C_VEL
LIN {X 0,Y 218.84,Z 714.27,A -85,B 0,C 180,E1 -21123.123,E2 -21123.123} C_VEL
LIN {X 0,Y 221.716,Z 655.889,A -85,B 0,C 180,E1 -21125.401,E2 -21125.401} C_VEL
LIN {X 0,Y 212.247,Z 632.614,A -85,B 0,C 180,E1 -21127.461,E2 -21127.461} C_VEL
LIN {X 0,Y 206.974,Z 620.539,A -85,B 0,C 180,E1 -21128.659,E2 -21128.659} C_VEL
LIN {X 0,Y 206.813,Z 619.725,A -85,B 0,C 180,E1 -21128.772,E2 -21128.772} C_VEL
LIN {X 0,Y 206.877,Z 619.718,A -85,B 0,C 180,E1 -21132.199,E2 -21132.199} C_VEL
LIN {X 0,Y 206.913,Z 619.713,A -85,B 0,C 180,E1 -21136.248,E2 -21136.248} C_VEL
LIN {X 0,Y 207.133,Z 619.685,A -85,B 0,C 180,E1 -21140.235,E2 -21140.235} C_VEL
LIN {X 0,Y 207.189,Z 619.678,A -85,B 0,C 180,E1 -21142.204,E2 -21142.204} C_VEL
LIN {X 0,Y 207.384,Z 619.653,A -85,B 0,C 180,E1 -21148.06,E2 -21148.06} C_VEL
LIN {X 0,Y 207.516,Z 619.635,A -85,B 0,C 180,E1 -21150.002,E2 -21150.002} C_VEL
LIN {X 0,Y 207.386,Z 619.651,A -85,B 0,C 180,E1 -21151.944,E2 -21151.944} C_VEL
LIN {X 0,Y 207.191,Z 619.674,A -85,B 0,C 180,E1 -21157.8,E2 -21157.8} C_VEL
LIN {X 0,Y 206.986,Z 619.698,A -85,B 0,C 180,E1 -21161.757,E2 -21161.757} C_VEL
LIN {X 0,Y 206.87,Z 619.713,A -85,B 0,C 180,E1 -21165.773,E2 -21165.773} C_VEL
LIN {X 0,Y 206.787,Z 619.711,A -85,B 0,C 180,E1 -21169.871,E2 -21169.871} C_VEL
LIN {X 0,Y 206.767,Z 619.726,A -85,B 0,C 180,E1 -21174.074,E2 -21174.074} C_VEL
LIN {X 0,Y 206.748,Z 619.729,A -85,B 0,C 180,E1 -21178.42,E2 -21178.42} C_VEL
LIN {X 0,Y 206.706,Z 619.719,A -85,B 0,C 180,E1 -21182.959,E2 -21182.959} C_VEL
LIN {X 0,Y 206.684,Z 619.732,A -85,B 0,C 180,E1 -21187.741,E2 -21187.741} C_VEL
LIN {X 0,Y 206.647,Z 619.743,A -85,B 0,C 180,E1 -21191.564,E2 -21191.564} C_VEL
LIN {X 0,Y 206.639,Z 619.74,A -85,B 0,C 180,E1 -21195.583,E2 -21195.583} C_VEL
LIN {X 0,Y 206.666,Z 619.723,A -85,B 0,C 180,E1 -21199.75,E2 -21199.75} C_VEL
LIN {X 0,Y 206.705,Z 619.716,A -85,B 0,C 180,E1 -21204.69,E2 -21204.69} C_VEL
LIN {X 0,Y 206.729,Z 619.729,A -85,B 0,C 180,E1 -21209.34,E2 -21209.34} C_VEL
LIN {X 0,Y 206.738,Z 619.734,A -85,B 0,C 180,E1 -21213.773,E2 -21213.773} C_VEL
LIN {X 0,Y 206.745,Z 619.724,A -85,B 0,C 180,E1 -21218.042,E2 -21218.042} C_VEL
LIN {X 0,Y 206.879,Z 619.691,A -85,B 0,C 180,E1 -21222.197,E2 -21222.197} C_VEL
LIN {X 0,Y 206.9,Z 619.697,A -85,B 0,C 180,E1 -21226.245,E2 -21226.245} C_VEL
LIN {X 0,Y 207.106,Z 619.685,A -85,B 0,C 180,E1 -21230.232,E2 -21230.232} C_VEL
LIN {X 0,Y 207.068,Z 619.692,A -85,B 0,C 180,E1 -21234.156,E2 -21234.156} C_VEL
LIN {X 0,Y 207.388,Z 619.645,A -85,B 0,C 180,E1 -21238.058,E2 -21238.058} C_VEL
LIN {X 0,Y 207.522,Z 619.622,A -85,B 0,C 180,E1 -21240,E2 -21240} C_VEL
LIN {X 0,Y 207.388,Z 619.633,A -85,B 0,C 180,E1 -21241.942,E2 -21241.942} C_VEL
LIN {X 0,Y 207.148,Z 619.679,A -85,B 0,C 180,E1 -21247.8,E2 -21247.8} C_VEL
LIN {X 0,Y 206.927,Z 619.707,A -85,B 0,C 180,E1 -21251.759,E2 -21251.759} C_VEL
LIN {X 0,Y 206.837,Z 619.709,A -85,B 0,C 180,E1 -21255.773,E2 -21255.773} C_VEL
LIN {X 0,Y 206.754,Z 619.731,A -85,B 0,C 180,E1 -21259.872,E2 -21259.872} C_VEL
LIN {X 0,Y 206.754,Z 619.729,A -85,B 0,C 180,E1 -21264.074,E2 -21264.074} C_VEL
LIN {X 0,Y 206.751,Z 619.732,A -85,B 0,C 180,E1 -21268.418,E2 -21268.418} C_VEL
LIN {X 0,Y 206.709,Z 619.734,A -85,B 0,C 180,E1 -21272.956,E2 -21272.956} C_VEL
LIN {X 0,Y 206.686,Z 619.738,A -85,B 0,C 180,E1 -21277.739,E2 -21277.739} C_VEL
LIN {X 0,Y 206.649,Z 619.745,A -85,B 0,C 180,E1 -21281.562,E2 -21281.562} C_VEL
LIN {X 0,Y 206.641,Z 619.746,A -85,B 0,C 180,E1 -21285.58,E2 -21285.58} C_VEL
LIN {X 0,Y 206.71,Z 619.737,A -85,B 0,C 180,E1 -21289.82,E2 -21289.82} C_VEL
LIN {X 0,Y 208.742,Z 628.896,A -85,B 0,C 180,E1 -21293.906,E2 -21293.906} C_VEL
LIN {X 0,Y 209.778,Z 633.909,A -85,B 0,C 180,E1 -21296.055,E2 -21296.055} C_VEL
LIN {X 0,Y 210.633,Z 635.267,A -85,B 0,C 180,E1 -21296.349,E2 -21296.349} C_VEL
LIN {X 0,Y 212.617,Z 638.698,A -85,B 0,C 180,E1 -21296.727,E2 -21296.727} C_VEL
LIN {X 0,Y 213.228,Z 642.045,A -85,B 0,C 180,E1 -21296.959,E2 -21296.959} C_VEL
LIN {X 0,Y 212.798,Z 644.984,A -85,B 0,C 180,E1 -21297.008,E2 -21297.008} C_VEL
LIN {X 0,Y 209.65,Z 652.055,A -85,B 0,C 180,E1 -21297.008,E2 -21297.008} C_VEL
LIN {X 0,Y 209.595,Z 654.494,A -85,B 0,C 180,E1 -21297.136,E2 -21297.136} C_VEL
LIN {X 0,Y 209.701,Z 654.819,A -85,B 0,C 180,E1 -21297.163,E2 -21297.163} C_VEL
LIN {X 0,Y 210.51,Z 660.634,A -85,B 0,C 180,E1 -21297.525,E2 -21297.525} C_VEL
LIN {X 0,Y 213.916,Z 693.32,A -85,B 0,C 180,E1 -21299.379,E2 -21299.379} C_VEL
LIN {X 0,Y 211.426,Z 743.142,A -85,B 0,C 180,E1 -21301.454,E2 -21301.454} C_VEL
LIN {X 0,Y 210.255,Z 756.626,A -85,B 0,C 180,E1 -21302.366,E2 -21302.366} C_VEL
LIN {X 0,Y 208.727,Z 768.517,A -85,B 0,C 180,E1 -21303.502,E2 -21303.502} C_VEL
LIN {X 0,Y 206.77,Z 781.06,A -85,B 0,C 180,E1 -21305.124,E2 -21305.124} C_VEL
LIN {X 0,Y 204.864,Z 792.371,A -85,B 0,C 180,E1 -21307.029,E2 -21307.029} C_VEL
LIN {X 0,Y 203.102,Z 802.232,A -85,B 0,C 180,E1 -21309.115,E2 -21309.115} C_VEL
LIN {X 0,Y 201.257,Z 811.903,A -85,B 0,C 180,E1 -21311.68,E2 -21311.68} C_VEL
LIN {X 0,Y 199.723,Z 820.949,A -85,B 0,C 180,E1 -21314.695,E2 -21314.695} C_VEL
LIN {X 0,Y 198.531,Z 828.121,A -85,B 0,C 180,E1 -21317.735,E2 -21317.735} C_VEL
LIN {X 0,Y 197.949,Z 833.824,A -85,B 0,C 180,E1 -21320.804,E2 -21320.804} C_VEL
LIN {X 0,Y 197.755,Z 838.788,A -85,B 0,C 180,E1 -21324.323,E2 -21324.323} C_VEL
LIN {X 0,Y 197.765,Z 840.538,A -85,B 0,C 180,E1 -21325.922,E2 -21325.922} C_VEL
LIN {X 0,Y 197.699,Z 842.337,A -85,B 0,C 180,E1 -21327.961,E2 -21327.961} C_VEL
LIN {X 0,Y 197.729,Z 843.64,A -85,B 0,C 180,E1 -21329.998,E2 -21329.998} C_VEL
LIN {X 0,Y 197.63,Z 844.501,A -85,B 0,C 180,E1 -21332.036,E2 -21332.036} C_VEL
LIN {X 0,Y 197.468,Z 844.992,A -85,B 0,C 180,E1 -21334.764,E2 -21334.764} C_VEL
LIN {X 0,Y 197.584,Z 844.579,A -85,B 0,C 180,E1 -21338.177,E2 -21338.177} C_VEL
LIN {X 0,Y 198.489,Z 842.628,A -85,B 0,C 180,E1 -21342.263,E2 -21342.263} C_VEL
LIN {X 0,Y 199.803,Z 840.097,A -85,B 0,C 180,E1 -21345.294,E2 -21345.294} C_VEL
LIN {X 0,Y 201.84,Z 836.632,A -85,B 0,C 180,E1 -21348.26,E2 -21348.26} C_VEL
LIN {X 0,Y 204.268,Z 832.138,A -85,B 0,C 180,E1 -21351.175,E2 -21351.175} C_VEL
LIN {X 0,Y 207.8,Z 825.455,A -85,B 0,C 180,E1 -21354.473,E2 -21354.473} C_VEL
LIN {X 0,Y 211.506,Z 818.285,A -85,B 0,C 180,E1 -21357.184,E2 -21357.184} C_VEL
LIN {X 0,Y 215.816,Z 809.481,A -85,B 0,C 180,E1 -21359.774,E2 -21359.774} C_VEL
LIN {X 0,Y 219.767,Z 800.595,A -85,B 0,C 180,E1 -21361.845,E2 -21361.845} C_VEL
LIN {X 0,Y 223.637,Z 790.97,A -85,B 0,C 180,E1 -21363.631,E2 -21363.631} C_VEL
LIN {X 0,Y 227.399,Z 780.587,A -85,B 0,C 180,E1 -21365.141,E2 -21365.141} C_VEL
LIN {X 0,Y 230.84,Z 769.457,A -85,B 0,C 180,E1 -21366.416,E2 -21366.416} C_VEL
LIN {X 0,Y 234.223,Z 756.094,A -85,B 0,C 180,E1 -21367.55,E2 -21367.55} C_VEL
LIN {X 0,Y 236.625,Z 743.556,A -85,B 0,C 180,E1 -21368.314,E2 -21368.314} C_VEL
LIN {X 0,Y 238.541,Z 727.005,A -85,B 0,C 180,E1 -21369.003,E2 -21369.003} C_VEL
LIN {X 0,Y 241.169,Z 699.169,A -85,B 0,C 180,E1 -21370.052,E2 -21370.052} C_VEL
LIN {X 0,Y 240.787,Z 688.904,A -85,B 0,C 180,E1 -21370.91,E2 -21370.91} C_VEL
LIN {X 0,Y 237.818,Z 680.729,A -85,B 0,C 180,E1 -21372.665,E2 -21372.665} C_VEL
LIN {X 0,Y 234.766,Z 673.601,A -85,B 0,C 180,E1 -21374.569,E2 -21374.569} C_VEL
LIN {X 0,Y 232.295,Z 668.4,A -85,B 0,C 180,E1 -21376.254,E2 -21376.254} C_VEL
LIN {X 0,Y 230.246,Z 664.257,A -85,B 0,C 180,E1 -21377.815,E2 -21377.815} C_VEL
LIN {X 0,Y 227.405,Z 658.778,A -85,B 0,C 180,E1 -21380.289,E2 -21380.289} C_VEL
LIN {X 0,Y 224.014,Z 652.613,A -85,B 0,C 180,E1 -21384.213,E2 -21384.213} C_VEL
LIN {X 0,Y 221.827,Z 649.14,A -85,B 0,C 180,E1 -21388.136,E2 -21388.136} C_VEL
LIN {X 0,Y 220.95,Z 647.106,A -85,B 0,C 180,E1 -21392.465,E2 -21392.465} C_VEL
LIN {X 0,Y 221.44,Z 646.911,A -85,B 0,C 180,E1 -21396.118,E2 -21396.118} C_VEL
LIN {X 0,Y 223.363,Z 648.197,A -85,B 0,C 180,E1 -21400.172,E2 -21400.172} C_VEL
LIN {X 0,Y 227.211,Z 652.875,A -85,B 0,C 180,E1 -21404.81,E2 -21404.81} C_VEL
LIN {X 0,Y 230.821,Z 657.585,A -85,B 0,C 180,E1 -21407.854,E2 -21407.854} C_VEL
LIN {X 0,Y 233.415,Z 661.68,A -85,B 0,C 180,E1 -21409.738,E2 -21409.738} C_VEL
LIN {X 0,Y 238.219,Z 669.439,A -85,B 0,C 180,E1 -21412.661,E2 -21412.661} C_VEL
LIN {X 0,Y 240.953,Z 674.891,A -85,B 0,C 180,E1 -21414.164,E2 -21414.164} C_VEL
LIN {X 0,Y 242.758,Z 679.35,A -85,B 0,C 180,E1 -21415.168,E2 -21415.168} C_VEL
LIN {X 0,Y 238.298,Z 724.233,A -85,B 0,C 180,E1 -21416.883,E2 -21416.883} C_VEL
LIN {X 0,Y 236.325,Z 736.996,A -85,B 0,C 180,E1 -21417.656,E2 -21417.656} C_VEL
LIN {X 0,Y 233.879,Z 749.018,A -85,B 0,C 180,E1 -21418.702,E2 -21418.702} C_VEL
LIN {X 0,Y 230.811,Z 760.449,A -85,B 0,C 180,E1 -21420,E2 -21420} C_VEL
LIN {X 0,Y 226.964,Z 772.34,A -85,B 0,C 180,E1 -21421.774,E2 -21421.774} C_VEL
LIN {X 0,Y 223.296,Z 782.049,A -85,B 0,C 180,E1 -21423.609,E2 -21423.609} C_VEL
LIN {X 0,Y 219.015,Z 791.609,A -85,B 0,C 180,E1 -21425.891,E2 -21425.891} C_VEL
LIN {X 0,Y 214.989,Z 799.703,A -85,B 0,C 180,E1 -21428.375,E2 -21428.375} C_VEL
LIN {X 0,Y 211.242,Z 806.467,A -85,B 0,C 180,E1 -21431.029,E2 -21431.029} C_VEL
LIN {X 0,Y 208.054,Z 811.741,A -85,B 0,C 180,E1 -21433.677,E2 -21433.677} C_VEL
LIN {X 0,Y 205.243,Z 816.058,A -85,B 0,C 180,E1 -21436.516,E2 -21436.516} C_VEL
LIN {X 0,Y 203.082,Z 819.047,A -85,B 0,C 180,E1 -21439.165,E2 -21439.165} C_VEL
LIN {X 0,Y 200.822,Z 821.733,A -85,B 0,C 180,E1 -21442.641,E2 -21442.641} C_VEL
LIN {X 0,Y 199.636,Z 822.778,A -85,B 0,C 180,E1 -21444.989,E2 -21444.989} C_VEL
LIN {X 0,Y 198.581,Z 823.344,A -85,B 0,C 180,E1 -21447.781,E2 -21447.781} C_VEL
LIN {X 0,Y 197.679,Z 822.901,A -85,B 0,C 180,E1 -21451.437,E2 -21451.437} C_VEL
LIN {X 0,Y 197.322,Z 821.228,A -85,B 0,C 180,E1 -21455.001,E2 -21455.001} C_VEL
LIN {X 0,Y 197.442,Z 818.394,A -85,B 0,C 180,E1 -21458.459,E2 -21458.459} C_VEL
LIN {X 0,Y 197.929,Z 814.439,A -85,B 0,C 180,E1 -21461.788,E2 -21461.788} C_VEL
LIN {X 0,Y 198.699,Z 809.253,A -85,B 0,C 180,E1 -21465.024,E2 -21465.024} C_VEL
LIN {X 0,Y 199.876,Z 801.949,A -85,B 0,C 180,E1 -21468.518,E2 -21468.518} C_VEL
LIN {X 0,Y 201.317,Z 794.223,A -85,B 0,C 180,E1 -21471.426,E2 -21471.426} C_VEL
LIN {X 0,Y 203.098,Z 784.856,A -85,B 0,C 180,E1 -21474.224,E2 -21474.224} C_VEL
LIN {X 0,Y 205.026,Z 774.325,A -85,B 0,C 180,E1 -21476.742,E2 -21476.742} C_VEL
LIN {X 0,Y 207.033,Z 762.792,A -85,B 0,C 180,E1 -21478.897,E2 -21478.897} C_VEL
LIN {X 0,Y 208.805,Z 750.306,A -85,B 0,C 180,E1 -21480.732,E2 -21480.732} C_VEL
LIN {X 0,Y 210.316,Z 737.752,A -85,B 0,C 180,E1 -21482.109,E2 -21482.109} C_VEL
LIN {X 0,Y 211.472,Z 724.172,A -85,B 0,C 180,E1 -21483.194,E2 -21483.194} C_VEL
LIN {X 0,Y 212.396,Z 708.673,A -85,B 0,C 180,E1 -21483.954,E2 -21483.954} C_VEL
LIN {X 0,Y 214.966,Z 657.329,A -85,B 0,C 180,E1 -21486.024,E2 -21486.024} C_VEL
LIN {X 0,Y 206.085,Z 635.502,A -85,B 0,C 180,E1 -21488.043,E2 -21488.043} C_VEL
LIN {X 0,Y 199.926,Z 621.549,A -85,B 0,C 180,E1 -21489.489,E2 -21489.489} C_VEL
LIN {X 0,Y 199.758,Z 620.604,A -85,B 0,C 180,E1 -21489.605,E2 -21489.605} C_VEL
LIN {X 0,Y 199.805,Z 620.594,A -85,B 0,C 180,E1 -21493.659,E2 -21493.659} C_VEL
LIN {X 0,Y 200.067,Z 620.562,A -85,B 0,C 180,E1 -21499.605,E2 -21499.605} C_VEL
LIN {X 0,Y 200.132,Z 620.557,A -85,B 0,C 180,E1 -21501.927,E2 -21501.927} C_VEL
LIN {X 0,Y 200.324,Z 620.532,A -85,B 0,C 180,E1 -21507.992,E2 -21507.992} C_VEL
LIN {X 0,Y 200.481,Z 620.512,A -85,B 0,C 180,E1 -21510.002,E2 -21510.002} C_VEL
LIN {X 0,Y 200.038,Z 620.566,A -85,B 0,C 180,E1 -21514.031,E2 -21514.031} C_VEL
LIN {X 0,Y 200.134,Z 620.553,A -85,B 0,C 180,E1 -21518.077,E2 -21518.077} C_VEL
LIN {X 0,Y 199.917,Z 620.579,A -85,B 0,C 180,E1 -21522.179,E2 -21522.179} C_VEL
LIN {X 0,Y 199.808,Z 620.594,A -85,B 0,C 180,E1 -21526.345,E2 -21526.345} C_VEL
LIN {X 0,Y 199.703,Z 620.596,A -85,B 0,C 180,E1 -21530.607,E2 -21530.607} C_VEL
LIN {X 0,Y 199.677,Z 620.613,A -85,B 0,C 180,E1 -21534.986,E2 -21534.986} C_VEL
LIN {X 0,Y 199.679,Z 620.606,A -85,B 0,C 180,E1 -21539.524,E2 -21539.524} C_VEL
LIN {X 0,Y 199.681,Z 620.597,A -85,B 0,C 180,E1 -21542.36,E2 -21542.36} C_VEL
LIN {X 0,Y 199.627,Z 620.605,A -85,B 0,C 180,E1 -21546.765,E2 -21546.765} C_VEL
LIN {X 0,Y 199.613,Z 620.616,A -85,B 0,C 180,E1 -21549.33,E2 -21549.33} C_VEL
LIN {X 0,Y 199.579,Z 620.621,A -85,B 0,C 180,E1 -21552.312,E2 -21552.312} C_VEL
LIN {X 0,Y 199.586,Z 620.621,A -85,B 0,C 180,E1 -21555.231,E2 -21555.231} C_VEL
LIN {X 0,Y 199.585,Z 620.611,A -85,B 0,C 180,E1 -21558.007,E2 -21558.007} C_VEL
LIN {X 0,Y 199.616,Z 620.598,A -85,B 0,C 180,E1 -21560.769,E2 -21560.769} C_VEL
LIN {X 0,Y 199.62,Z 620.603,A -85,B 0,C 180,E1 -21565.715,E2 -21565.715} C_VEL
LIN {X 0,Y 199.708,Z 620.602,A -85,B 0,C 180,E1 -21568.139,E2 -21568.139} C_VEL
LIN {X 0,Y 199.692,Z 620.609,A -85,B 0,C 180,E1 -21572.773,E2 -21572.773} C_VEL
LIN {X 0,Y 199.721,Z 620.602,A -85,B 0,C 180,E1 -21577.227,E2 -21577.227} C_VEL
LIN {X 0,Y 199.802,Z 620.574,A -85,B 0,C 180,E1 -21581.76,E2 -21581.76} C_VEL
LIN {X 0,Y 199.84,Z 620.571,A -85,B 0,C 180,E1 -21585.749,E2 -21585.749} C_VEL
LIN {X 0,Y 200.03,Z 620.563,A -85,B 0,C 180,E1 -21589.882,E2 -21589.882} C_VEL
LIN {X 0,Y 200.03,Z 620.569,A -85,B 0,C 180,E1 -21593.95,E2 -21593.95} C_VEL
LIN {X 0,Y 200.328,Z 620.524,A -85,B 0,C 180,E1 -21597.99,E2 -21597.99} C_VEL
LIN {X 0,Y 200.486,Z 620.497,A -85,B 0,C 180,E1 -21600,E2 -21600} C_VEL
LIN {X 0,Y 200.034,Z 620.556,A -85,B 0,C 180,E1 -21604.03,E2 -21604.03} C_VEL
LIN {X 0,Y 200.097,Z 620.559,A -85,B 0,C 180,E1 -21608.077,E2 -21608.077} C_VEL
LIN {X 0,Y 199.876,Z 620.586,A -85,B 0,C 180,E1 -21612.18,E2 -21612.18} C_VEL
LIN {X 0,Y 199.773,Z 620.591,A -85,B 0,C 180,E1 -21616.346,E2 -21616.346} C_VEL
LIN {X 0,Y 199.679,Z 620.616,A -85,B 0,C 180,E1 -21620.608,E2 -21620.608} C_VEL
LIN {X 0,Y 199.671,Z 620.608,A -85,B 0,C 180,E1 -21624.985,E2 -21624.985} C_VEL
LIN {X 0,Y 199.682,Z 620.613,A -85,B 0,C 180,E1 -21629.521,E2 -21629.521} C_VEL
LIN {X 0,Y 199.684,Z 620.61,A -85,B 0,C 180,E1 -21632.358,E2 -21632.358} C_VEL
LIN {X 0,Y 199.63,Z 620.619,A -85,B 0,C 180,E1 -21636.762,E2 -21636.762} C_VEL
LIN {X 0,Y 199.615,Z 620.621,A -85,B 0,C 180,E1 -21639.327,E2 -21639.327} C_VEL
LIN {X 0,Y 199.581,Z 620.626,A -85,B 0,C 180,E1 -21642.309,E2 -21642.309} C_VEL
LIN {X 0,Y 199.587,Z 620.626,A -85,B 0,C 180,E1 -21645.228,E2 -21645.228} C_VEL
LIN {X 0,Y 199.654,Z 620.645,A -85,B 0,C 180,E1 -21649.263,E2 -21649.263} C_VEL
LIN {X 0,Y 201.796,Z 630.219,A -85,B 0,C 180,E1 -21653.694,E2 -21653.694} C_VEL
LIN {X 0,Y 202.542,Z 633.869,A -85,B 0,C 180,E1 -21655.314,E2 -21655.314} C_VEL
LIN {X 0,Y 209.701,Z 654.819,A -85,B 0,C 180,E1 -21657.163,E2 -21657.163} C_VEL
LIN {X 0,Y 210.532,Z 658.466,A -85,B 0,C 180,E1 -21657.426,E2 -21657.426} C_VEL
LIN {X 0,Y 210.268,Z 664.26,A -85,B 0,C 180,E1 -21657.67,E2 -21657.67} C_VEL
LIN {X 0,Y 206.574,Z 679.986,A -85,B 0,C 180,E1 -21658.021,E2 -21658.021} C_VEL
LIN {X 0,Y 206.421,Z 685.957,A -85,B 0,C 180,E1 -21658.288,E2 -21658.288} C_VEL
LIN {X 0,Y 207.215,Z 694.778,A -85,B 0,C 180,E1 -21658.784,E2 -21658.784} C_VEL
LIN {X 0,Y 204.69,Z 742.696,A -85,B 0,C 180,E1 -21660.846,E2 -21660.846} C_VEL
LIN {X 0,Y 203.489,Z 756.175,A -85,B 0,C 180,E1 -21661.786,E2 -21661.786} C_VEL
LIN {X 0,Y 201.767,Z 769.103,A -85,B 0,C 180,E1 -21663.073,E2 -21663.073} C_VEL
LIN {X 0,Y 199.782,Z 781.404,A -85,B 0,C 180,E1 -21664.75,E2 -21664.75} C_VEL
LIN {X 0,Y 197.839,Z 792.586,A -85,B 0,C 180,E1 -21666.719,E2 -21666.719} C_VEL
LIN {X 0,Y 195.962,Z 802.722,A -85,B 0,C 180,E1 -21668.981,E2 -21668.981} C_VEL
LIN {X 0,Y 194.171,Z 811.898,A -85,B 0,C 180,E1 -21671.534,E2 -21671.534} C_VEL
LIN {X 0,Y 192.607,Z 820.872,A -85,B 0,C 180,E1 -21674.658,E2 -21674.658} C_VEL
LIN {X 0,Y 191.429,Z 827.964,A -85,B 0,C 180,E1 -21677.811,E2 -21677.811} C_VEL
LIN {X 0,Y 190.926,Z 832.789,A -85,B 0,C 180,E1 -21680.463,E2 -21680.463} C_VEL
LIN {X 0,Y 190.705,Z 838.091,A -85,B 0,C 180,E1 -21684.285,E2 -21684.285} C_VEL
LIN {X 0,Y 190.711,Z 839.701,A -85,B 0,C 180,E1 -21685.771,E2 -21685.771} C_VEL
LIN {X 0,Y 190.638,Z 841.574,A -85,B 0,C 180,E1 -21687.885,E2 -21687.885} C_VEL
LIN {X 0,Y 190.66,Z 842.986,A -85,B 0,C 180,E1 -21689.998,E2 -21689.998} C_VEL
LIN {X 0,Y 190.56,Z 843.909,A -85,B 0,C 180,E1 -21692.111,E2 -21692.111} C_VEL
LIN {X 0,Y 190.4,Z 844.486,A -85,B 0,C 180,E1 -21694.708,E2 -21694.708} C_VEL
LIN {X 0,Y 190.526,Z 844.238,A -85,B 0,C 180,E1 -21698.483,E2 -21698.483} C_VEL
LIN {X 0,Y 191.515,Z 842.433,A -85,B 0,C 180,E1 -21702.717,E2 -21702.717} C_VEL
LIN {X 0,Y 192.35,Z 840.955,A -85,B 0,C 180,E1 -21704.816,E2 -21704.816} C_VEL
LIN {X 0,Y 194.311,Z 837.954,A -85,B 0,C 180,E1 -21707.902,E2 -21707.902} C_VEL
LIN {X 0,Y 196.705,Z 833.96,A -85,B 0,C 180,E1 -21710.931,E2 -21710.931} C_VEL
LIN {X 0,Y 199.738,Z 828.84,A -85,B 0,C 180,E1 -21713.906,E2 -21713.906} C_VEL
LIN {X 0,Y 203.242,Z 822.676,A -85,B 0,C 180,E1 -21716.711,E2 -21716.711} C_VEL
LIN {X 0,Y 207.467,Z 815.016,A -85,B 0,C 180,E1 -21719.416,E2 -21719.416} C_VEL
LIN {X 0,Y 212.15,Z 805.585,A -85,B 0,C 180,E1 -21722.006,E2 -21722.006} C_VEL
LIN {X 0,Y 216.922,Z 794.997,A -85,B 0,C 180,E1 -21724.256,E2 -21724.256} C_VEL
LIN {X 0,Y 221.252,Z 784.346,A -85,B 0,C 180,E1 -21725.988,E2 -21725.988} C_VEL
LIN {X 0,Y 225.306,Z 772.534,A -85,B 0,C 180,E1 -21727.461,E2 -21727.461} C_VEL
LIN {X 0,Y 229.074,Z 759.292,A -85,B 0,C 180,E1 -21728.687,E2 -21728.687} C_VEL
LIN {X 0,Y 231.922,Z 745.712,A -85,B 0,C 180,E1 -21729.59,E2 -21729.59} C_VEL
LIN {X 0,Y 233.982,Z 731.172,A -85,B 0,C 180,E1 -21730.239,E2 -21730.239} C_VEL
LIN {X 0,Y 237.084,Z 700.429,A -85,B 0,C 180,E1 -21731.415,E2 -21731.415} C_VEL
LIN {X 0,Y 236.881,Z 692.359,A -85,B 0,C 180,E1 -21732.121,E2 -21732.121} C_VEL
LIN {X 0,Y 233.736,Z 683.443,A -85,B 0,C 180,E1 -21734.162,E2 -21734.162} C_VEL
LIN {X 0,Y 230.111,Z 675.011,A -85,B 0,C 180,E1 -21736.725,E2 -21736.725} C_VEL
LIN {X 0,Y 227.773,Z 670.058,A -85,B 0,C 180,E1 -21738.652,E2 -21738.652} C_VEL
LIN {X 0,Y 225.292,Z 664.973,A -85,B 0,C 180,E1 -21741.028,E2 -21741.028} C_VEL
LIN {X 0,Y 222.368,Z 659.239,A -85,B 0,C 180,E1 -21744.718,E2 -21744.718} C_VEL
LIN {X 0,Y 220.394,Z 655.946,A -85,B 0,C 180,E1 -21748.604,E2 -21748.604} C_VEL
LIN {X 0,Y 219.724,Z 654.183,A -85,B 0,C 180,E1 -21752.299,E2 -21752.299} C_VEL
LIN {X 0,Y 219.756,Z 653.849,A -85,B 0,C 180,E1 -21753.563,E2 -21753.563} C_VEL
LIN {X 0,Y 220.728,Z 654.197,A -85,B 0,C 180,E1 -21757.537,E2 -21757.537} C_VEL
LIN {X 0,Y 222.112,Z 655.403,A -85,B 0,C 180,E1 -21760.228,E2 -21760.228} C_VEL
LIN {X 0,Y 225.365,Z 659.394,A -85,B 0,C 180,E1 -21764.288,E2 -21764.288} C_VEL
LIN {X 0,Y 228.746,Z 664.05,A -85,B 0,C 180,E1 -21767.33,E2 -21767.33} C_VEL
LIN {X 0,Y 231.217,Z 668.238,A -85,B 0,C 180,E1 -21769.251,E2 -21769.251} C_VEL
LIN {X 0,Y 235.407,Z 675.242,A -85,B 0,C 180,E1 -21771.941,E2 -21771.941} C_VEL
LIN {X 0,Y 237.716,Z 680.15,A -85,B 0,C 180,E1 -21773.319,E2 -21773.319} C_VEL
LIN {X 0,Y 238.609,Z 682.521,A -85,B 0,C 180,E1 -21773.856,E2 -21773.856} C_VEL
LIN {X 0,Y 234.108,Z 724.898,A -85,B 0,C 180,E1 -21775.502,E2 -21775.502} C_VEL
LIN {X 0,Y 231.946,Z 738.029,A -85,B 0,C 180,E1 -21776.318,E2 -21776.318} C_VEL
LIN {X 0,Y 229.094,Z 750.932,A -85,B 0,C 180,E1 -21777.472,E2 -21777.472} C_VEL
LIN {X 0,Y 225.686,Z 762.782,A -85,B 0,C 180,E1 -21778.875,E2 -21778.875} C_VEL
LIN {X 0,Y 222.102,Z 773.129,A -85,B 0,C 180,E1 -21780.453,E2 -21780.453} C_VEL
LIN {X 0,Y 218.051,Z 783.147,A -85,B 0,C 180,E1 -21782.407,E2 -21782.407} C_VEL
LIN {X 0,Y 213.522,Z 792.563,A -85,B 0,C 180,E1 -21784.72,E2 -21784.72} C_VEL
LIN {X 0,Y 209.279,Z 800.57,A -85,B 0,C 180,E1 -21787.234,E2 -21787.234} C_VEL
LIN {X 0,Y 204.714,Z 808.179,A -85,B 0,C 180,E1 -21790.383,E2 -21790.383} C_VEL
LIN {X 0,Y 201.074,Z 813.617,A -85,B 0,C 180,E1 -21793.386,E2 -21793.386} C_VEL
LIN {X 0,Y 197.975,Z 817.876,A -85,B 0,C 180,E1 -21796.576,E2 -21796.576} C_VEL
LIN {X 0,Y 195.012,Z 821.386,A -85,B 0,C 180,E1 -21800.453,E2 -21800.453} C_VEL
LIN {X 0,Y 192.821,Z 823.298,A -85,B 0,C 180,E1 -21804.333,E2 -21804.333} C_VEL
LIN {X 0,Y 191.232,Z 823.803,A -85,B 0,C 180,E1 -21808.539,E2 -21808.539} C_VEL
LIN {X 0,Y 190.486,Z 823.019,A -85,B 0,C 180,E1 -21811.947,E2 -21811.947} C_VEL
LIN {X 0,Y 190.203,Z 820.974,A -85,B 0,C 180,E1 -21815.624,E2 -21815.624} C_VEL
LIN {X 0,Y 190.401,Z 817.775,A -85,B 0,C 180,E1 -21819.186,E2 -21819.186} C_VEL
LIN {X 0,Y 190.999,Z 813.443,A -85,B 0,C 180,E1 -21822.619,E2 -21822.619} C_VEL
LIN {X 0,Y 191.819,Z 808.027,A -85,B 0,C 180,E1 -21825.886,E2 -21825.886} C_VEL
LIN {X 0,Y 192.966,Z 801.383,A -85,B 0,C 180,E1 -21829.04,E2 -21829.04} C_VEL
LIN {X 0,Y 194.507,Z 793.216,A -85,B 0,C 180,E1 -21832.106,E2 -21832.106} C_VEL
LIN {X 0,Y 196.285,Z 784.259,A -85,B 0,C 180,E1 -21834.809,E2 -21834.809} C_VEL
LIN {X 0,Y 198.226,Z 773.872,A -85,B 0,C 180,E1 -21837.322,E2 -21837.322} C_VEL
LIN {X 0,Y 200.305,Z 762.132,A -85,B 0,C 180,E1 -21839.546,E2 -21839.546} C_VEL
LIN {X 0,Y 201.995,Z 750.62,A -85,B 0,C 180,E1 -21841.266,E2 -21841.266} C_VEL
LIN {X 0,Y 203.518,Z 738.209,A -85,B 0,C 180,E1 -21842.671,E2 -21842.671} C_VEL
LIN {X 0,Y 204.737,Z 724.458,A -85,B 0,C 180,E1 -21843.802,E2 -21843.802} C_VEL
LIN {X 0,Y 205.704,Z 708.674,A -85,B 0,C 180,E1 -21844.595,E2 -21844.595} C_VEL
LIN {X 0,Y 208.351,Z 659.091,A -85,B 0,C 180,E1 -21846.653,E2 -21846.653} C_VEL
LIN {X 0,Y 199.561,Z 637.48,A -85,B 0,C 180,E1 -21848.74,E2 -21848.74} C_VEL
LIN {X 0,Y 192.831,Z 622.08,A -85,B 0,C 180,E1 -21850.398,E2 -21850.398} C_VEL
LIN {X 0,Y 192.729,Z 621.476,A -85,B 0,C 180,E1 -21850.463,E2 -21850.463} C_VEL
LIN {X 0,Y 192.772,Z 621.471,A -85,B 0,C 180,E1 -21855.217,E2 -21855.217} C_VEL
LIN {X 0,Y 193.019,Z 621.44,A -85,B 0,C 180,E1 -21859.513,E2 -21859.513} C_VEL
LIN {X 0,Y 193.006,Z 621.444,A -85,B 0,C 180,E1 -21863.731,E2 -21863.731} C_VEL
LIN {X 0,Y 193.266,Z 621.411,A -85,B 0,C 180,E1 -21867.918,E2 -21867.918} C_VEL
LIN {X 0,Y 193.445,Z 621.389,A -85,B 0,C 180,E1 -21870.002,E2 -21870.002} C_VEL
LIN {X 0,Y 192.985,Z 621.446,A -85,B 0,C 180,E1 -21874.179,E2 -21874.179} C_VEL
LIN {X 0,Y 193.081,Z 621.433,A -85,B 0,C 180,E1 -21878.374,E2 -21878.374} C_VEL
LIN {X 0,Y 192.856,Z 621.461,A -85,B 0,C 180,E1 -21882.632,E2 -21882.632} C_VEL
LIN {X 0,Y 192.761,Z 621.469,A -85,B 0,C 180,E1 -21886.961,E2 -21886.961} C_VEL
LIN {X 0,Y 192.64,Z 621.482,A -85,B 0,C 180,E1 -21891.399,E2 -21891.399} C_VEL
LIN {X 0,Y 192.668,Z 621.482,A -85,B 0,C 180,E1 -21894.227,E2 -21894.227} C_VEL
LIN {X 0,Y 192.654,Z 621.484,A -85,B 0,C 180,E1 -21898.894,E2 -21898.894} C_VEL
LIN {X 0,Y 192.603,Z 621.471,A -85,B 0,C 180,E1 -21903.187,E2 -21903.187} C_VEL
LIN {X 0,Y 192.556,Z 621.491,A -85,B 0,C 180,E1 -21908.353,E2 -21908.353} C_VEL
LIN {X 0,Y 192.518,Z 621.503,A -85,B 0,C 180,E1 -21913.104,E2 -21913.104} C_VEL
LIN {X 0,Y 192.497,Z 621.5,A -85,B 0,C 180,E1 -21916.906,E2 -21916.906} C_VEL
LIN {X 0,Y 192.557,Z 621.468,A -85,B 0,C 180,E1 -21921.65,E2 -21921.65} C_VEL
LIN {X 0,Y 192.605,Z 621.48,A -85,B 0,C 180,E1 -21926.816,E2 -21926.816} C_VEL
LIN {X 0,Y 192.671,Z 621.486,A -85,B 0,C 180,E1 -21931.693,E2 -21931.693} C_VEL
LIN {X 0,Y 192.691,Z 621.478,A -85,B 0,C 180,E1 -21936.347,E2 -21936.347} C_VEL
LIN {X 0,Y 192.737,Z 621.455,A -85,B 0,C 180,E1 -21941.46,E2 -21941.46} C_VEL
LIN {X 0,Y 192.768,Z 621.449,A -85,B 0,C 180,E1 -21945.214,E2 -21945.214} C_VEL
LIN {X 0,Y 192.952,Z 621.443,A -85,B 0,C 180,E1 -21949.567,E2 -21949.567} C_VEL
LIN {X 0,Y 192.992,Z 621.444,A -85,B 0,C 180,E1 -21953.728,E2 -21953.728} C_VEL
LIN {X 0,Y 193.27,Z 621.403,A -85,B 0,C 180,E1 -21957.916,E2 -21957.916} C_VEL
LIN {X 0,Y 193.45,Z 621.372,A -85,B 0,C 180,E1 -21960,E2 -21960} C_VEL
LIN {X 0,Y 192.98,Z 621.435,A -85,B 0,C 180,E1 -21964.177,E2 -21964.177} C_VEL
LIN {X 0,Y 193.044,Z 621.439,A -85,B 0,C 180,E1 -21968.374,E2 -21968.374} C_VEL
LIN {X 0,Y 192.801,Z 621.463,A -85,B 0,C 180,E1 -21972.634,E2 -21972.634} C_VEL
LIN {X 0,Y 192.727,Z 621.474,A -85,B 0,C 180,E1 -21976.962,E2 -21976.962} C_VEL
LIN {X 0,Y 192.616,Z 621.493,A -85,B 0,C 180,E1 -21981.4,E2 -21981.4} C_VEL
LIN {X 0,Y 192.654,Z 621.486,A -85,B 0,C 180,E1 -21984.213,E2 -21984.213} C_VEL
LIN {X 0,Y 192.657,Z 621.49,A -85,B 0,C 180,E1 -21988.891,E2 -21988.891} C_VEL
LIN {X 0,Y 192.606,Z 621.49,A -85,B 0,C 180,E1 -21993.185,E2 -21993.185} C_VEL
LIN {X 0,Y 192.558,Z 621.499,A -85,B 0,C 180,E1 -21998.351,E2 -21998.351} C_VEL
LIN {X 0,Y 192.498,Z 621.51,A -85,B 0,C 180,E1 -22003.095,E2 -22003.095} C_VEL
LIN {X 0,Y 192.592,Z 621.561,A -85,B 0,C 180,E1 -22008.696,E2 -22008.696} C_VEL
LIN {X 0,Y 194.449,Z 629.805,A -85,B 0,C 180,E1 -22012.67,E2 -22012.67} C_VEL
LIN {X 0,Y 195.259,Z 633.643,A -85,B 0,C 180,E1 -22014.376,E2 -22014.376} C_VEL
LIN {X 0,Y 203.583,Z 657.774,A -85,B 0,C 180,E1 -22016.615,E2 -22016.615} C_VEL
LIN {X 0,Y 206.421,Z 685.957,A -85,B 0,C 180,E1 -22018.288,E2 -22018.288} C_VEL
LIN {X 0,Y 206.136,Z 689.835,A -85,B 0,C 180,E1 -22018.44,E2 -22018.44} C_VEL
LIN {X 0,Y 203.633,Z 696.048,A -85,B 0,C 180,E1 -22018.472,E2 -22018.472} C_VEL
LIN {X 0,Y 200.776,Z 702.281,A -85,B 0,C 180,E1 -22018.475,E2 -22018.475} C_VEL
LIN {X 0,Y 199.978,Z 706.23,A -85,B 0,C 180,E1 -22018.585,E2 -22018.585} C_VEL
LIN {X 0,Y 197.89,Z 743.228,A -85,B 0,C 180,E1 -22020.256,E2 -22020.256} C_VEL
LIN {X 0,Y 196.584,Z 757.127,A -85,B 0,C 180,E1 -22021.286,E2 -22021.286} C_VEL
LIN {X 0,Y 194.82,Z 769.618,A -85,B 0,C 180,E1 -22022.614,E2 -22022.614} C_VEL
LIN {X 0,Y 192.782,Z 781.706,A -85,B 0,C 180,E1 -22024.345,E2 -22024.345} C_VEL
LIN {X 0,Y 190.811,Z 792.737,A -85,B 0,C 180,E1 -22026.385,E2 -22026.385} C_VEL
LIN {X 0,Y 188.742,Z 803.56,A -85,B 0,C 180,E1 -22028.949,E2 -22028.949} C_VEL
LIN {X 0,Y 186.779,Z 813.474,A -85,B 0,C 180,E1 -22031.913,E2 -22031.913} C_VEL
LIN {X 0,Y 185.23,Z 821.961,A -85,B 0,C 180,E1 -22035.158,E2 -22035.158} C_VEL
LIN {X 0,Y 184.215,Z 828.766,A -85,B 0,C 180,E1 -22038.444,E2 -22038.444} C_VEL
LIN {X 0,Y 183.756,Z 833.327,A -85,B 0,C 180,E1 -22041.198,E2 -22041.198} C_VEL
LIN {X 0,Y 183.662,Z 837.326,A -85,B 0,C 180,E1 -22044.222,E2 -22044.222} C_VEL
LIN {X 0,Y 183.578,Z 840.778,A -85,B 0,C 180,E1 -22047.804,E2 -22047.804} C_VEL
LIN {X 0,Y 183.592,Z 842.279,A -85,B 0,C 180,E1 -22049.998,E2 -22049.998} C_VEL
LIN {X 0,Y 183.49,Z 843.315,A -85,B 0,C 180,E1 -22052.193,E2 -22052.193} C_VEL
LIN {X 0,Y 183.324,Z 843.918,A -85,B 0,C 180,E1 -22054.618,E2 -22054.618} C_VEL
LIN {X 0,Y 183.492,Z 843.849,A -85,B 0,C 180,E1 -22058.81,E2 -22058.81} C_VEL
LIN {X 0,Y 183.916,Z 843.258,A -85,B 0,C 180,E1 -22061.012,E2 -22061.012} C_VEL
LIN {X 0,Y 185.465,Z 840.847,A -85,B 0,C 180,E1 -22065.38,E2 -22065.38} C_VEL
LIN {X 0,Y 188.356,Z 836.853,A -85,B 0,C 180,E1 -22069.619,E2 -22069.619} C_VEL
LIN {X 0,Y 191.117,Z 832.704,A -85,B 0,C 180,E1 -22072.711,E2 -22072.711} C_VEL
LIN {X 0,Y 195.005,Z 826.494,A -85,B 0,C 180,E1 -22076.196,E2 -22076.196} C_VEL
LIN {X 0,Y 199.087,Z 819.781,A -85,B 0,C 180,E1 -22079.035,E2 -22079.035} C_VEL
LIN {X 0,Y 203.773,Z 811.626,A -85,B 0,C 180,E1 -22081.73,E2 -22081.73} C_VEL
LIN {X 0,Y 208.033,Z 803.429,A -85,B 0,C 180,E1 -22083.875,E2 -22083.875} C_VEL
LIN {X 0,Y 212.655,Z 793.576,A -85,B 0,C 180,E1 -22085.914,E2 -22085.914} C_VEL
LIN {X 0,Y 217.221,Z 782.63,A -85,B 0,C 180,E1 -22087.636,E2 -22087.636} C_VEL
LIN {X 0,Y 221.47,Z 770.635,A -85,B 0,C 180,E1 -22089.099,E2 -22089.099} C_VEL
LIN {X 0,Y 225.132,Z 758.162,A -85,B 0,C 180,E1 -22090.223,E2 -22090.223} C_VEL
LIN {X 0,Y 228.105,Z 744.645,A -85,B 0,C 180,E1 -22091.102,E2 -22091.102} C_VEL
LIN {X 0,Y 230.136,Z 730.76,A -85,B 0,C 180,E1 -22091.724,E2 -22091.724} C_VEL
LIN {X 0,Y 233.211,Z 701.911,A -85,B 0,C 180,E1 -22092.817,E2 -22092.817} C_VEL
LIN {X 0,Y 233.119,Z 696.019,A -85,B 0,C 180,E1 -22093.34,E2 -22093.34} C_VEL
LIN {X 0,Y 230.658,Z 688.516,A -85,B 0,C 180,E1 -22095.145,E2 -22095.145} C_VEL
LIN {X 0,Y 227.566,Z 680.731,A -85,B 0,C 180,E1 -22097.563,E2 -22097.563} C_VEL
LIN {X 0,Y 225.478,Z 676.122,A -85,B 0,C 180,E1 -22099.392,E2 -22099.392} C_VEL
LIN {X 0,Y 223.34,Z 671.361,A -85,B 0,C 180,E1 -22101.652,E2 -22101.652} C_VEL
LIN {X 0,Y 220.734,Z 665.893,A -85,B 0,C 180,E1 -22105.23,E2 -22105.23} C_VEL
LIN {X 0,Y 219.084,Z 662.898,A -85,B 0,C 180,E1 -22108.757,E2 -22108.757} C_VEL
LIN {X 0,Y 218.466,Z 661.003,A -85,B 0,C 180,E1 -22112.877,E2 -22112.877} C_VEL
LIN {X 0,Y 219.052,Z 661.003,A -85,B 0,C 180,E1 -22116.494,E2 -22116.494} C_VEL
LIN {X 0,Y 220.571,Z 662.149,A -85,B 0,C 180,E1 -22119.803,E2 -22119.803} C_VEL
LIN {X 0,Y 223.655,Z 666.199,A -85,B 0,C 180,E1 -22123.908,E2 -22123.908} C_VEL
LIN {X 0,Y 226.659,Z 670.548,A -85,B 0,C 180,E1 -22126.785,E2 -22126.785} C_VEL
LIN {X 0,Y 228.778,Z 674.178,A -85,B 0,C 180,E1 -22128.499,E2 -22128.499} C_VEL
LIN {X 0,Y 232.679,Z 681.056,A -85,B 0,C 180,E1 -22131.207,E2 -22131.207} C_VEL
LIN {X 0,Y 234.585,Z 685.495,A -85,B 0,C 180,E1 -22132.477,E2 -22132.477} C_VEL
LIN {X 0,Y 230.205,Z 725.324,A -85,B 0,C 180,E1 -22134.046,E2 -22134.046} C_VEL
LIN {X 0,Y 228.041,Z 737.926,A -85,B 0,C 180,E1 -22134.814,E2 -22134.814} C_VEL
LIN {X 0,Y 225.487,Z 749.344,A -85,B 0,C 180,E1 -22135.817,E2 -22135.817} C_VEL
LIN {X 0,Y 222.225,Z 760.479,A -85,B 0,C 180,E1 -22137.054,E2 -22137.054} C_VEL
LIN {X 0,Y 217.903,Z 772.544,A -85,B 0,C 180,E1 -22138.845,E2 -22138.845} C_VEL
LIN {X 0,Y 213.799,Z 782.368,A -85,B 0,C 180,E1 -22140.706,E2 -22140.706} C_VEL
LIN {X 0,Y 209.374,Z 791.46,A -85,B 0,C 180,E1 -22142.885,E2 -22142.885} C_VEL
LIN {X 0,Y 204.712,Z 799.713,A -85,B 0,C 180,E1 -22145.4,E2 -22145.4} C_VEL
LIN {X 0,Y 200.51,Z 806.45,A -85,B 0,C 180,E1 -22148.059,E2 -22148.059} C_VEL
LIN {X 0,Y 196.117,Z 812.861,A -85,B 0,C 180,E1 -22151.367,E2 -22151.367} C_VEL
LIN {X 0,Y 192.315,Z 817.683,A -85,B 0,C 180,E1 -22154.821,E2 -22154.821} C_VEL
LIN {X 0,Y 190.226,Z 820.12,A -85,B 0,C 180,E1 -22157.191,E2 -22157.191} C_VEL
LIN {X 0,Y 187.716,Z 822.585,A -85,B 0,C 180,E1 -22160.62,E2 -22160.62} C_VEL
LIN {X 0,Y 185.553,Z 824.064,A -85,B 0,C 180,E1 -22164.636,E2 -22164.636} C_VEL
LIN {X 0,Y 184.096,Z 824.156,A -85,B 0,C 180,E1 -22168.599,E2 -22168.599} C_VEL
LIN {X 0,Y 183.308,Z 822.979,A -85,B 0,C 180,E1 -22172.496,E2 -22172.496} C_VEL
LIN {X 0,Y 183.101,Z 820.613,A -85,B 0,C 180,E1 -22176.293,E2 -22176.293} C_VEL
LIN {X 0,Y 183.411,Z 817.066,A -85,B 0,C 180,E1 -22179.976,E2 -22179.976} C_VEL
LIN {X 0,Y 184.056,Z 812.382,A -85,B 0,C 180,E1 -22183.494,E2 -22183.494} C_VEL
LIN {X 0,Y 185.169,Z 805.674,A -85,B 0,C 180,E1 -22187.316,E2 -22187.316} C_VEL
LIN {X 0,Y 186.482,Z 798.567,A -85,B 0,C 180,E1 -22190.484,E2 -22190.484} C_VEL
LIN {X 0,Y 188.183,Z 790.002,A -85,B 0,C 180,E1 -22193.518,E2 -22193.518} C_VEL
LIN {X 0,Y 190.19,Z 780.05,A -85,B 0,C 180,E1 -22196.341,E2 -22196.341} C_VEL
LIN {X 0,Y 192.166,Z 769.35,A -85,B 0,C 180,E1 -22198.752,E2 -22198.752} C_VEL
LIN {X 0,Y 194.154,Z 757.861,A -85,B 0,C 180,E1 -22200.791,E2 -22200.791} C_VEL
LIN {X 0,Y 195.827,Z 746.148,A -85,B 0,C 180,E1 -22202.424,E2 -22202.424} C_VEL
LIN {X 0,Y 197.327,Z 732.888,A -85,B 0,C 180,E1 -22203.792,E2 -22203.792} C_VEL
LIN {X 0,Y 198.406,Z 719.137,A -85,B 0,C 180,E1 -22204.781,E2 -22204.781} C_VEL
LIN {X 0,Y 201.635,Z 660.603,A -85,B 0,C 180,E1 -22207.346,E2 -22207.346} C_VEL
LIN {X 0,Y 192.834,Z 638.983,A -85,B 0,C 180,E1 -22209.507,E2 -22209.507} C_VEL
LIN {X 0,Y 185.799,Z 622.787,A -85,B 0,C 180,E1 -22211.336,E2 -22211.336} C_VEL
LIN {X 0,Y 185.754,Z 622.346,A -85,B 0,C 180,E1 -22211.424,E2 -22211.424} C_VEL
LIN {X 0,Y 185.765,Z 622.345,A -85,B 0,C 180,E1 -22216.882,E2 -22216.882} C_VEL
LIN {X 0,Y 186.029,Z 622.313,A -85,B 0,C 180,E1 -22221.311,E2 -22221.311} C_VEL
LIN {X 0,Y 186.21,Z 622.29,A -85,B 0,C 180,E1 -22227.839,E2 -22227.839} C_VEL
LIN {X 0,Y 186.408,Z 622.265,A -85,B 0,C 180,E1 -22230.002,E2 -22230.002} C_VEL
LIN {X 0,Y 185.932,Z 622.325,A -85,B 0,C 180,E1 -22234.338,E2 -22234.338} C_VEL
LIN {X 0,Y 186.031,Z 622.313,A -85,B 0,C 180,E1 -22238.694,E2 -22238.694} C_VEL
LIN {X 0,Y 185.768,Z 622.345,A -85,B 0,C 180,E1 -22243.122,E2 -22243.122} C_VEL
LIN {X 0,Y 185.678,Z 622.342,A -85,B 0,C 180,E1 -22248.869,E2 -22248.869} C_VEL
LIN {X 0,Y 185.604,Z 622.364,A -85,B 0,C 180,E1 -22254.664,E2 -22254.664} C_VEL
LIN {X 0,Y 185.583,Z 622.361,A -85,B 0,C 180,E1 -22259.495,E2 -22259.495} C_VEL
LIN {X 0,Y 185.504,Z 622.352,A -85,B 0,C 180,E1 -22264.634,E2 -22264.634} C_VEL
LIN {X 0,Y 185.51,Z 622.366,A -85,B 0,C 180,E1 -22267.315,E2 -22267.315} C_VEL
LIN {X 0,Y 185.476,Z 622.377,A -85,B 0,C 180,E1 -22270.727,E2 -22270.727} C_VEL
LIN {X 0,Y 185.468,Z 622.378,A -85,B 0,C 180,E1 -22273.948,E2 -22273.948} C_VEL
LIN {X 0,Y 185.476,Z 622.362,A -85,B 0,C 180,E1 -22279.277,E2 -22279.277} C_VEL
LIN {X 0,Y 185.511,Z 622.341,A -85,B 0,C 180,E1 -22282.713,E2 -22282.713} C_VEL
LIN {X 0,Y 185.553,Z 622.364,A -85,B 0,C 180,E1 -22287.977,E2 -22287.977} C_VEL
LIN {X 0,Y 185.588,Z 622.364,A -85,B 0,C 180,E1 -22290.577,E2 -22290.577} C_VEL
LIN {X 0,Y 185.586,Z 622.367,A -85,B 0,C 180,E1 -22295.383,E2 -22295.383} C_VEL
LIN {X 0,Y 185.68,Z 622.336,A -85,B 0,C 180,E1 -22301.136,E2 -22301.136} C_VEL
LIN {X 0,Y 185.7,Z 622.327,A -85,B 0,C 180,E1 -22304.638,E2 -22304.638} C_VEL
LIN {X 0,Y 185.896,Z 622.321,A -85,B 0,C 180,E1 -22309.418,E2 -22309.418} C_VEL
LIN {X 0,Y 185.955,Z 622.32,A -85,B 0,C 180,E1 -22313.49,E2 -22313.49} C_VEL
LIN {X 0,Y 186.214,Z 622.282,A -85,B 0,C 180,E1 -22317.837,E2 -22317.837} C_VEL
LIN {X 0,Y 186.414,Z 622.247,A -85,B 0,C 180,E1 -22320,E2 -22320} C_VEL
LIN {X 0,Y 185.926,Z 622.313,A -85,B 0,C 180,E1 -22324.336,E2 -22324.336} C_VEL
LIN {X 0,Y 185.991,Z 622.317,A -85,B 0,C 180,E1 -22328.694,E2 -22328.694} C_VEL
LIN {X 0,Y 185.726,Z 622.342,A -85,B 0,C 180,E1 -22333.123,E2 -22333.123} C_VEL
LIN {X 0,Y 185.663,Z 622.354,A -85,B 0,C 180,E1 -22337.628,E2 -22337.628} C_VEL
LIN {X 0,Y 185.581,Z 622.371,A -85,B 0,C 180,E1 -22342.254,E2 -22342.254} C_VEL
LIN {X 0,Y 185.568,Z 622.37,A -85,B 0,C 180,E1 -22347.032,E2 -22347.032} C_VEL
LIN {X 0,Y 185.586,Z 622.369,A -85,B 0,C 180,E1 -22349.492,E2 -22349.492} C_VEL
LIN {X 0,Y 185.506,Z 622.377,A -85,B 0,C 180,E1 -22354.631,E2 -22354.631} C_VEL
LIN {X 0,Y 185.512,Z 622.378,A -85,B 0,C 180,E1 -22357.312,E2 -22357.312} C_VEL
LIN {X 0,Y 185.478,Z 622.384,A -85,B 0,C 180,E1 -22360.724,E2 -22360.724} C_VEL
LIN {X 0,Y 185.467,Z 622.384,A -85,B 0,C 180,E1 -22366.053,E2 -22366.053} C_VEL
LIN {X 0,Y 185.555,Z 622.579,A -85,B 0,C 180,E1 -22368.151,E2 -22368.151} C_VEL
LIN {X 0,Y 187.295,Z 630.241,A -85,B 0,C 180,E1 -22372,E2 -22372} C_VEL
LIN {X 0,Y 187.92,Z 633.07,A -85,B 0,C 180,E1 -22373.367,E2 -22373.367} C_VEL
LIN {X 0,Y 196.367,Z 657.528,A -85,B 0,C 180,E1 -22375.741,E2 -22375.741} C_VEL
LIN {X 0,Y 197.25,Z 661.277,A -85,B 0,C 180,E1 -22376.039,E2 -22376.039} C_VEL
LIN {X 0,Y 200.572,Z 694.764,A -85,B 0,C 180,E1 -22378.085,E2 -22378.085} C_VEL
LIN {X 0,Y 199.978,Z 706.23,A -85,B 0,C 180,E1 -22378.585,E2 -22378.585} C_VEL
LIN {X 0,Y 199.121,Z 712.026,A -85,B 0,C 180,E1 -22378.778,E2 -22378.778} C_VEL
LIN {X 0,Y 192.75,Z 730.784,A -85,B 0,C 180,E1 -22379.058,E2 -22379.058} C_VEL
LIN {X 0,Y 191.64,Z 736.563,A -85,B 0,C 180,E1 -22379.265,E2 -22379.265} C_VEL
LIN {X 0,Y 190.363,Z 751.149,A -85,B 0,C 180,E1 -22380.179,E2 -22380.179} C_VEL
LIN {X 0,Y 188.997,Z 762.466,A -85,B 0,C 180,E1 -22381.241,E2 -22381.241} C_VEL
LIN {X 0,Y 186.996,Z 775.308,A -85,B 0,C 180,E1 -22382.887,E2 -22382.887} C_VEL
LIN {X 0,Y 184.798,Z 787.561,A -85,B 0,C 180,E1 -22384.968,E2 -22384.968} C_VEL
LIN {X 0,Y 182.653,Z 798.442,A -85,B 0,C 180,E1 -22387.368,E2 -22387.368} C_VEL
LIN {X 0,Y 180.678,Z 808.274,A -85,B 0,C 180,E1 -22390.099,E2 -22390.099} C_VEL
LIN {X 0,Y 179.106,Z 816.343,A -85,B 0,C 180,E1 -22392.882,E2 -22392.882} C_VEL
LIN {X 0,Y 177.697,Z 824.177,A -85,B 0,C 180,E1 -22396.27,E2 -22396.27} C_VEL
LIN {X 0,Y 176.906,Z 830.435,A -85,B 0,C 180,E1 -22399.699,E2 -22399.699} C_VEL
LIN {X 0,Y 176.608,Z 835.34,A -85,B 0,C 180,E1 -22403.141,E2 -22403.141} C_VEL
LIN {X 0,Y 176.539,Z 839.009,A -85,B 0,C 180,E1 -22406.574,E2 -22406.574} C_VEL
LIN {X 0,Y 176.526,Z 841.544,A -85,B 0,C 180,E1 -22409.998,E2 -22409.998} C_VEL
LIN {X 0,Y 176.42,Z 842.659,A -85,B 0,C 180,E1 -22412.281,E2 -22412.281} C_VEL
LIN {X 0,Y 176.262,Z 843.342,A -85,B 0,C 180,E1 -22414.571,E2 -22414.571} C_VEL
LIN {X 0,Y 176.447,Z 843.453,A -85,B 0,C 180,E1 -22419.165,E2 -22419.165} C_VEL
LIN {X 0,Y 177.608,Z 842.041,A -85,B 0,C 180,E1 -22423.732,E2 -22423.732} C_VEL
LIN {X 0,Y 178.607,Z 840.757,A -85,B 0,C 180,E1 -22425.986,E2 -22425.986} C_VEL
